# B&R Automation Studio project Nitto (part 14)

#### FB_WebbufferCtrl.st
```iecst
(********************************************************************
 * COPYRIGHT -- Microsoft
 ********************************************************************
 * Programm: MAIN
 * Datei: FB_WebbufferCtrl.st
 * Autor: awalz
 * Erstellt: 26. Juni 2014
 ********************************************************************
 * Implementierung des Programms MAIN
 ********************************************************************)

(* TODO: Bitte Kommentar hier einfügen *)
FUNCTION_BLOCK FB_WebbufferCtrl
	axis.bufferaxis(machineaxis := machineaxis, data := data, CONST := CONST, dancer := dancer, tensionoffset := torqueoffset);
	axis.refSwitchConfig(Enable := TRUE, Axis := axis.ctrl.AxisREF);
//	machineaxis();
	dancer();
	axis.ctrl();
	emcy_inputs();
	keys(clk := clk);
	torqueoffset(enable := TRUE, limitvisuneg := -50, limitvisupos := 50);

//	IF (keys.up.LDT.rtrig.Q OR keys.down.LDT.rtrig.Q ) AND axis.bufferaxis.MC_BR_VelocityControl_0.Active THEN
//		axis.bufferaxis.cmd := CONST.AXIS.STOP;(*deaktivierung des FBs Torque*)
//	ELSIF machineaxis.MC_ReadStatus_0.ContinuousMotion THEN
//		axis.bufferaxis.cmd := CONST.AXIS.START;
//	END_IF
	(*aufruf der Action *)

	status.ready := (axis.ctrl.MC_ReadStatus_0.ContinuousMotion OR axis.ctrl.MC_ReadStatus_0.SynchronizedMotion
				OR axis.ctrl.MC_ReadStatus_0.StandStill) AND NOT axis.ctrl.MC_ReadStatus_0.Disabled;
	status(axisState := axis.ctrl.MC_ReadStatus_0);
	IF axis.ctrl.BasicControl.AxisState.Homed AND (axis.ctrl.MC_ReadStatus_0.StandStill OR axis.ctrl.MC_ReadStatus_0.ContinuousMotion) THEN
		keys.home.LDT.aktion := CONST.LAMP.ON;
	ELSIF axis.ctrl.MC_ReadStatus_0.Disabled THEN
		keys.home.LDT.aktion := CONST.LAMP.BLINK1000;
	ELSIF axis.ctrl.MC_ReadStatus_0.Errorstop THEN
		keys.home.LDT.aktion := CONST.LAMP.BLINK200;
	END_IF
	IF axis.ctrl.MC_ReadStatus_0.Errorstop  AND keys.up.LDT.button AND keys.down.LDT.button THEN
		axis.ctrl(cmd := CONST.AXIS.RESET);
	END_IF
	IF (NOT emcy_inputs.EMCY_Door1 OR NOT emcy_inputs.EMCY_Door2 OR NOT emcy_inputs.EMCY_Door3 OR NOT safety.RequestSTO
		OR NOT emcy_inputs.EMCY_Door4 OR NOT emcy_inputs.EMCY_Door5 OR NOT emcy_inputs.EMCY_Door6) AND NOT  axis.ctrl.MC_ReadStatus_0.Disabled THEN
		axis.ctrl(cmd := CONST.AXIS.POWER_OFF);
		axis.bufferaxis.cmd := CONST.AXIS.STOP;
		mechbrakeON_OFF := FALSE;
	ELSIF  emcy_inputs.EMCY_Door1 AND emcy_inputs.EMCY_Door2 AND emcy_inputs.EMCY_Door3 AND emcy_inputs.EMCY_Door4 AND
		emcy_inputs.EMCY_Door5 AND emcy_inputs.EMCY_Door6 AND axis.ctrl.MC_ReadStatus_0.Disabled AND safety.RequestSTO THEN
		axis.ctrl(cmd := CONST.AXIS.POWER_ON);
		mechbrakeON_OFF := TRUE;

	END_IF
	(* Signal um zu Joggen siehe Mastermodul ac_manual*)
	IF emcy_inputs.EMCY_Door1 AND emcy_inputs.EMCY_Door2 AND emcy_inputs.EMCY_Door3 AND emcy_inputs.EMCY_Door4 AND
		emcy_inputs.EMCY_Door5 AND emcy_inputs.EMCY_Door6 THEN
		emcy_inputs.EMCY_DoorsClosed := TRUE;
	ELSE
		emcy_inputs.EMCY_DoorsClosed := FALSE;
	END_IF

CASE StateCtrl OF
	CTRL_FIRST_START:
		busy := TRUE;
		(*axis.bufferaxis.*)
		StateCtrl := CTRL_EMERGENCYSTOP_BEFORE;

	CTRL_MANUAL_BEFORE://10

		IF BetrCtrl.value = CONST.MACHINEMODES.MANUAL THEN
			BetrStatus(set := TRUE,value := CONST.MACHINEMODES.MANUAL);
			busy := FALSE;
			err(reset := TRUE);
			timer(IN:= FALSE);
			state := ST_IDLE;
			firstStart := TRUE;
			brakeholddelay(PT := T#2s);
			IF axis.ctrl.MC_ReadStatus_0.StandStill THEN
				brakeholddelay.IN:= TRUE;
			END_IF

			IF brakeholddelay.Q AND NOT mechbrakeON_OFF THEN
				brakeholddelay(IN:= FALSE);
				mechbrakeON_OFF := TRUE;
				StateCtrl := CTRL_MANUAL;
			ELSIF mechbrakeON_OFF THEN//25.03.15
				StateCtrl := CTRL_MANUAL;
			END_IF
		ELSIF BetrCtrl.value = CONST.MACHINEMODES.EMERGENCYSTOP THEN
			StateCtrl := CTRL_EMERGENCYSTOP_BEFORE;
		ELSIF BetrCtrl.value = CONST.MACHINEMODES.SAFETYSTOP THEN
			StateCtrl := CTRL_SAFETYSTOP_BEFORE;
		ELSIF BetrCtrl.value = CONST.MACHINEMODES.AUTOMATIC THEN
			StateCtrl := CTRL_AUTO_BEFORE;
		END_IF

	CTRL_MANUAL:
		IF BetrCtrl.value <> CONST.MACHINEMODES.MANUAL THEN
			err(reset := TRUE);
			busy := TRUE;
			StateCtrl := CTRL_MANUAL_AFTER;
		ELSE
			ac_manualbufferCtrl;
			IF axis.ctrl.BasicControl.AxisState.Homed THEN
				 acBuffercyclic; (* Aufruf der Aktion nur wenn die Achse referenziert ist 04.12.14*)
			END_IF
		END_IF

	CTRL_MANUAL_AFTER:

		 acSetModeAfterBuffer;

	CTRL_AUTO_BEFORE:
		IF BetrCtrl.value = CONST.MACHINEMODES.AUTOMATIC THEN
			BetrStatus(set := TRUE, value := CONST.MACHINEMODES.AUTOMATIC);
			(*clamp.init(clk := clk);
			chkStatus.enable := TRUE;*)
			err(reset := TRUE);
			busy := FALSE;
			state := ST_IDLE;
			brakeholddelay(PT := T#2s);
			IF axis.ctrl.MC_ReadStatus_0.StandStill THEN
				brakeholddelay.IN:= TRUE;
			END_IF
			IF brakeholddelay.Q AND NOT mechbrakeON_OFF THEN
				brakeholddelay(IN:= FALSE);
				mechbrakeON_OFF := TRUE;
				StateCtrl := CTRL_AUTO;
			ELSIF mechbrakeON_OFF THEN//25.03.15
				StateCtrl := CTRL_AUTO;
			END_IF
		ELSIF BetrCtrl.value = CONST.MACHINEMODES.EMERGENCYSTOP THEN
			StateCtrl := CTRL_EMERGENCYSTOP_BEFORE;
		ELSIF BetrCtrl.value = CONST.MACHINEMODES.SAFETYSTOP THEN
			StateCtrl := CTRL_SAFETYSTOP_BEFORE;
		ELSIF BetrCtrl.value = CONST.MACHINEMODES.MANUAL THEN
			StateCtrl := CTRL_MANUAL_BEFORE;
		END_IF

	(* ******************************** *)
	(* *********** AUTO *************** *)
	(* ******************************** *)
	CTRL_AUTO:
		IF BetrCtrl.value <> CONST.MACHINEMODES.AUTOMATIC THEN
			err(reset := TRUE);
			busy := TRUE;
			StateCtrl := CTRL_AUTO_AFTER;
		ELSE
			IF axis.ctrl.BasicControl.AxisState.Homed THEN
				 acBuffercyclic; (* Aufruf der Aktion nur wenn die Achse referenziert ist 04.12.14*)
			END_IF
			(*ac_automatic();*)
		END_IF

	CTRL_AUTO_AFTER:
		(*chkStatus.enable := FALSE;*)
		acSetModeAfterBuffer;

	CTRL_STOP_BEFORE:
		IF BetrCtrl.value = CONST.MACHINEMODES.EMERGENCYSTOP THEN
			StateCtrl := CTRL_EMERGENCYSTOP_BEFORE;
		ELSIF BetrCtrl.value = CONST.MACHINEMODES.SAFETYSTOP THEN
			StateCtrl := CTRL_SAFETYSTOP_BEFORE;
		ELSE
			state := ST_IDLE;
			StateCtrl := CTRL_STOP;
		END_IF

	CTRL_STOP:
		IF BetrCtrl.value = CONST.MACHINEMODES.EMERGENCYSTOP THEN
			StateCtrl := CTRL_EMERGENCYSTOP_BEFORE;
		ELSIF BetrCtrl.value = CONST.MACHINEMODES.SAFETYSTOP THEN
			StateCtrl := CTRL_SAFETYSTOP_BEFORE;
		ELSE
			CASE state OF
			ST_IDLE:
				state := ST_QUIT;

			ST_QUIT:
				state := ST_IDLE;
				StateCtrl := CTRL_STOP_AFTER;
			END_CASE
		END_IF

	CTRL_STOP_AFTER:
		IF BetrCtrl.value = CONST.MACHINEMODES.EMERGENCYSTOP THEN
			StateCtrl := CTRL_EMERGENCYSTOP_BEFORE;
		ELSIF BetrCtrl.value = CONST.MACHINEMODES.SAFETYSTOP THEN
			StateCtrl := CTRL_SAFETYSTOP_BEFORE;
		ELSIF BetrCtrl.value = CONST.MACHINEMODES.MANUAL THEN
			StateCtrl := CTRL_MANUAL_BEFORE;
		ELSIF BetrCtrl.value = CONST.MACHINEMODES.AUTOMATIC THEN
			StateCtrl := CTRL_AUTO_BEFORE;
		END_IF

	CTRL_RESET_START:
		BetrStatus.set := TRUE;
		BetrStatus.value := CONST.MACHINEMODES.RESET;
		IF BetrCtrl.value = CONST.MACHINEMODES.EMERGENCYSTOP THEN
			StateCtrl := CTRL_EMERGENCYSTOP_BEFORE;
		ELSIF BetrCtrl.value = CONST.MACHINEMODES.SAFETYSTOP THEN
			StateCtrl := CTRL_SAFETYSTOP_BEFORE;
		ELSE
			IF axis.ctrl.busy  OR axis.ctrl.cmd <> CONST.AXIS.NOACTION THEN
			(*	axis.ctrl(cmd := CONST.AXIS.NOACTION);*)
			ELSE
				mechbrakeON_OFF := FALSE;
				axis.ctrl(cmd := CONST.AXIS.RESET);
				StateCtrl := CTRL_RESET;
			END_IF
		END_IF

	CTRL_RESET:
		axis.ctrl();
		IF BetrCtrl.value = CONST.MACHINEMODES.EMERGENCYSTOP THEN
			StateCtrl := CTRL_EMERGENCYSTOP_BEFORE;
		ELSIF BetrCtrl.value = CONST.MACHINEMODES.SAFETYSTOP THEN
			StateCtrl := CTRL_SAFETYSTOP_BEFORE;
		ELSE
			(*IF NOT unwinderaxis.busy THEN*)
				mechbrakeON_OFF := FALSE;

				axis.ctrl(cmd := CONST.AXIS.POWER_OFF);
				StateCtrl := CTRL_RESET_AFTER;
			(*END_IF*)
		END_IF

	CTRL_RESET_AFTER:
		IF BetrCtrl.value = CONST.MACHINEMODES.RESET THEN
			busy := FALSE;
		ELSE
			busy := TRUE;
			(*clamp.init(clk := clk);
			err.reset();*)
			err(reset := TRUE);
			IF BetrCtrl.value = CONST.MACHINEMODES.EMERGENCYSTOP THEN
				StateCtrl := CTRL_EMERGENCYSTOP_BEFORE;
			ELSIF BetrCtrl.value = CONST.MACHINEMODES.SAFETYSTOP THEN
				StateCtrl := CTRL_SAFETYSTOP_BEFORE;
			ELSIF BetrCtrl.value = CONST.MACHINEMODES.MANUAL THEN
				supplydelay(IN:= TRUE, PT := T#8s);
				IF supplydelay.Q THEN
					axis.ctrl(cmd := CONST.AXIS.POWER_ON);
					busy := TRUE;
					supplydelay(IN:= FALSE);
					StateCtrl := CTRL_MANUAL_BEFORE;
				END_IF
			ELSIF BetrCtrl.value = CONST.MACHINEMODES.AUTOMATIC THEN
				supplydelay(IN:= TRUE, PT := T#8s);
				IF supplydelay.Q THEN
					axis.ctrl(cmd := CONST.AXIS.POWER_ON);
					busy := TRUE;
					supplydelay(IN:= FALSE);
					StateCtrl := CTRL_AUTO_BEFORE;
				END_IF
			END_IF
		END_IF

	CTRL_SAFETYSTOP_BEFORE:
		IF BetrCtrl.value = CONST.MACHINEMODES.EMERGENCYSTOP THEN
			StateCtrl := CTRL_EMERGENCYSTOP_BEFORE;
		ELSE
//			BetrStatus.set := TRUE;
//			BetrStatus.value := CONST.MACHINEMODES.SAFETYSTOP;
//			mechbrakeON_OFF := FALSE;
//			axis.ctrl(cmd := CONST.AXIS.POWER_OFF);(* neue weil die Achse nicht ausgeschaltet wird*)
//			mechbrakeON_OFF := FALSE;
//			state := ST_IDLE;
//			StateCtrl := CTRL_SAFETYSTOP;
			mechbrakeON_OFF := FALSE;
			BetrStatus(set := TRUE,value := CONST.MACHINEMODES.SAFETYSTOP);
			state := ST_IDLE;
			axis.bufferaxis.cmd := CONST.AXIS.STOP;
			axis.ctrl.verzoegerung := 42000.0;
			axis.ctrl.cmd := CONST.AXIS.STOP;
			StateCtrl := CTRL_SAFETYSTOP;
		END_IF

	CTRL_SAFETYSTOP:
		IF BetrCtrl.value = CONST.MACHINEMODES.EMERGENCYSTOP THEN
			StateCtrl := CTRL_EMERGENCYSTOP_BEFORE;
		ELSE
//			CASE state OF
//			ST_IDLE:
//				mechbrakeON_OFF := FALSE;
//			(*	axis.ctrl.cmd := CONST.AXIS.RESET;*)
//				state := ST_QUIT;
//			ST_QUIT:
//				state := ST_QUIT;
//			(*	axis.ctrl(cmd := CONST.AXIS.RESET);*)
//				StateCtrl := CTRL_SAFETYSTOP_AFTER;
//			END_CASE
			IF axis.bufferaxis.MC_ReadStatus_0.StandStill OR axis.bufferaxis.MC_ReadStatus_0.Disabled  THEN
				axis.ctrl.cmd := CONST.AXIS.POWER_OFF;
				StateCtrl := CTRL_SAFETYSTOP_AFTER;
			END_IF
		END_IF

	CTRL_SAFETYSTOP_AFTER:
		busy := FALSE;
		IF BetrCtrl.value = CONST.MACHINEMODES.EMERGENCYSTOP THEN
			busy := TRUE;
			StateCtrl := CTRL_EMERGENCYSTOP_BEFORE;
		ELSIF BetrCtrl.value = CONST.MACHINEMODES.MANUAL THEN
			supplydelay(IN:= TRUE, PT := T#8s);
				IF supplydelay.Q THEN
					axis.ctrl(cmd := CONST.AXIS.POWER_ON);
					busy := TRUE;
					supplydelay(IN:= FALSE);
					StateCtrl := CTRL_MANUAL_BEFORE;
				END_IF
		ELSIF BetrCtrl.value = CONST.MACHINEMODES.AUTOMATIC THEN
				supplydelay(IN:= TRUE, PT := T#8s);
				IF supplydelay.Q THEN
					axis.ctrl(cmd := CONST.AXIS.POWER_ON);
					busy := TRUE;
					supplydelay(IN:= FALSE);
					StateCtrl := CTRL_AUTO_BEFORE;
				END_IF
		END_IF

	CTRL_EMERGENCYSTOP_BEFORE:
//		axis.ctrl(cmd := CONST.AXIS.RESET);
//		mechbrakeON_OFF := FALSE;
//		BetrStatus(set := TRUE,value := CONST.MACHINEMODES.EMERGENCYSTOP);
//		busy := FALSE;
//		StateCtrl := CTRL_EMERGENCYSTOP;
		BetrStatus(set := TRUE,value := CONST.MACHINEMODES.EMERGENCYSTOP);
		mechbrakeON_OFF := FALSE;
		axis.ctrl.verzoegerung:= 1666666; (*200m/min in 2 sek*)
		axis.ctrl.cmd := CONST.AXIS.STOP;
		StateCtrl := CTRL_EMERGENCYSTOP;

	CTRL_EMERGENCYSTOP:
		IF BetrCtrl.value = CONST.MACHINEMODES.EMERGENCYSTOP THEN
			IF axis.ctrl.MC_ReadStatus_0.StandStill OR axis.ctrl.MC_ReadStatus_0.Disabled  THEN
				axis.ctrl.cmd := CONST.AXIS.POWER_OFF;
			END_IF
		ELSE
			busy := TRUE;
			timer(IN := TRUE, PT := T#2s);
			StateCtrl := CTRL_EMERGENCYSTOP_AFTER;
		END_IF

	CTRL_EMERGENCYSTOP_AFTER:
		timer();
		IF BetrCtrl.value = CONST.MACHINEMODES.EMERGENCYSTOP THEN
			timer(IN := FALSE);
			BetrStatus(set := TRUE,value := CONST.MACHINEMODES.EMERGENCYSTOP);
			busy := FALSE;
			StateCtrl := CTRL_EMERGENCYSTOP;
		ELSIF timer.Q THEN
			timer(IN := FALSE);
			StateCtrl := CTRL_RESET_START;
		END_IF

	ELSE
		;
	END_CASE
END_FUNCTION_BLOCK
```

#### FB_WEBBUFFER.st
```iecst
(********************************************************************
 * COPYRIGHT -- Microsoft
 ********************************************************************
 * Programm: MAIN
 * Datei: FB_WEBBUFFER.st
 * Autor: awalz
 * Erstellt: 26. Juni 2014
 ********************************************************************
 * Implementierung des Programms MAIN
 ********************************************************************)

(* TODO: Bitte Kommentar hier einfügen *)
FUNCTION_BLOCK FB_WEBBUFFER
END_FUNCTION_BLOCK
```

#### FB_Bufferaxis.st
```iecst
(********************************************************************
 * COPYRIGHT -- Microsoft
 ********************************************************************
 * Programm: MAIN
 * Datei: NeuerFunktionsBlock.st
 * Autor: awalz
 * Erstellt: 10. Juli 2014
 ********************************************************************
 * Implementierung des Programms MAIN
 ********************************************************************)

(* TODO: Bitte Kommentar hier einfügen *)
FUNCTION_BLOCK FB_Bufferaxis
END_FUNCTION_BLOCK
```

#### FB_BufferConfig.st
```iecst
(********************************************************************
 * COPYRIGHT -- Microsoft
 ********************************************************************
 * Programm: MAIN
 * Datei: FB_BufferConfig.st
 * Autor: awalz
 * Erstellt: 10. Juli 2014
 ********************************************************************
 * Implementierung des Programms MAIN
 ********************************************************************)

(* TODO: Bitte Kommentar hier einfügen *)
FUNCTION_BLOCK FB_BufferConfig

		(*axis.refSwitchConfig(Enable := TRUE, Axis := axis.ctrl.AxisREF);*)
		axis.ctrl.BasicControl.Parameter.Deceleration := 1000;
		axis.ctrl.BasicControl.Parameter.Acceleration := 1000;
		pAxis ACCESS axis.ctrl.AxisREF;
		axis.ctrl();

CASE state OF
	ST_IDLE:
		IF cmd <> CONST.CUTTINGUNIT.CMDs.NO_CMD THEN
			busy := TRUE;
			err(reset := TRUE);
			cmdtmp := cmd;
			IF cmd = CONST.CUTTINGUNIT.CMDs.ABORT THEN
				state := ST_ABORT;
			ELSE
				IF cmd = CONST.CUTTINGUNIT.CMDs.CALIBR THEN
					state := ST_INIT_START;
				ELSIF cmd = CONST.CUTTINGUNIT.CMDs.MOVEFW OR cmd = CONST.CUTTINGUNIT.CMDs.MOVEBW THEN
					state := ST_MOVE_START;
//				ELSE
//					busy := FALSE;
//					err.reset();
				END_IF
			END_IF
		END_IF
//

	(*ST_SET_MODULO:*)

	ST_INIT_START:
		axis();
		IF NOT axis.ctrl.MC_ReadStatus_0.Disabled THEN
			axis.ctrl.cmd := CONST.AXIS.POWER_OFF;
		ELSE
			axis.ctrl.cmd := CONST.AXIS.NOACTION;
			IF NOT axis.ctrl.busy AND  axis.ctrl.MC_ReadStatus_0.Disabled THEN
				pAxis.dig_in.level.neg_hw_end := ncACTIV_HI + ncFORCE;
				pAxis.dig_in.level.pos_hw_end := ncACTIV_HI + ncFORCE;
				InitAxisSubjectPar.Axis := axis.ctrl.AxisREF;
				InitAxisSubjectPar.Subject := ncDIG_IN;
				InitAxisSubjectPar.Execute := TRUE;
				InitAxisSubjectPar();
				IF InitAxisSubjectPar.Done THEN
				(*	axis.refSwitchConfig(Enable := TRUE);*)
				(*	axis.refSwitchConfig.Axis := axis.ctrl.AxisREF;*)
					InitAxisSubjectPar.Execute := FALSE;
					state := ST_REF_START;
				ELSIF InitAxisSubjectPar.Error THEN
					err.text := 'Parameter ncDIG_IN nicht initialisiert';
					err.state := state;
					state := ST_ERROR;
				END_IF
			END_IF
		END_IF

	ST_REF_START:
		InitAxisSubjectPar();
		(*axis.refSwitchConfig();*)
		IF axis.ctrl.MC_ReadStatus_0.Disabled THEN
			axis.ctrl.cmd := CONST.AXIS.POWER_ON;
		ELSIF NOT axis.ctrl.busy AND axis.ctrl.MC_ReadStatus_0.StandStill THEN
		(*	axis.refSwitchConfig(Enable := TRUE);*)
			axis.ctrl.BasicControl.Parameter.HomeMode := mcHOME_LIMIT_SWITCH;
			axis.ctrl.cmd := CONST.AXIS.CALIBR; (* Achse referenzieren*)
			state := ST_CALIBR_WAIT;
		END_IF

	ST_CALIBR_WAIT:
	(*	axis.refSwitchConfig();*)
		IF axis.ctrl.BasicControl.AxisState.Homed THEN
			(*axis.refSwitchConfig(Enable := FALSE);*)
			cmd := CONST.CUTTINGUNIT.CMDs.NO_CMD;
			axis.ctrl(cmd := CONST.AXIS.NOACTION);
			status.ready := TRUE;
			cmdtmp := cmd;
			state := ST_QUIT;(* Achse ist referenziert*)
		(*	state := ST_CALIBR_START_NULLPOS;*)
		ELSIF cmd <> CONST.CUTTINGUNIT.CMDs.CALIBR THEN
			axis.ctrl(cmd := CONST.AXIS.STOP);
			state := ST_QUIT;
		END_IF

	ST_MOVE_START:
//		masterAxis.ctrl.ref.ReadStatus();
		IF cmd = CONST.CUTTINGUNIT.CMDs.NO_CMD THEN
			busy := FALSE;
			state := ST_IDLE;
		ELSE
			IF cmd = CONST.CUTTINGUNIT.CMDs.MOVEBW THEN
				axis.ctrl.velocity	:= 0.01;
				axis.ctrl.cmd := CONST.AXIS.JOG_NEG;
				state := ST_MOVE_WAIT;
			ELSE
				axis.ctrl.velocity := 0.02;
				axis.ctrl.cmd := CONST.AXIS.JOG_POS;
				state := ST_MOVE_WAIT;
			END_IF

		END_IF

	ST_MOVE_WAIT:
		axis.ctrl();
		IF cmd = CONST.CUTTINGUNIT.CMDs.NO_CMD THEN
			axis.ctrl(cmd := CONST.AXIS.NOACTION );
			state := ST_MOVE_QUIT;
		END_IF
//
	ST_MOVE_QUIT: (* hier evtl. koppeln*)
		state := ST_QUIT;

	ST_ERROR:
		IF LEN(err.fnc) < 1 THEN
			err.fnc := 'FB_CuttingConfig';
		END_IF
		err(flag := TRUE);
		state := ST_QUIT;

	ST_ABORT:
		state := ST_ABORT_QUIT;

	ST_ABORT_QUIT:
		busy := FALSE;
		IF cmd <> CONST.CUTTINGUNIT.CMDs.NO_CMD THEN
			state := ST_IDLE;
		END_IF

	ST_QUIT:
		IF cmd = CONST.CUTTINGUNIT.CMDs.ABORT THEN
			busy := TRUE;
			state := ST_ABORT;
		ELSE
			busy := FALSE;
			IF cmd = CONST.CUTTINGUNIT.CMDs.NO_CMD THEN
				axis.ctrl(cmd := CONST.AXIS.NOACTION);
				state := ST_IDLE;
			END_IF
		END_IF

	END_CASE
//InitAxisSubjectPar();
END_FUNCTION_BLOCK
```

#### FB_TorqueAxis.st
```iecst
(********************************************************************
 * COPYRIGHT -- Microsoft
 ********************************************************************
 * Programm: MAIN
 * Datei: FB_TorqueAxis.st
 * Autor: awalz
 * Erstellt: 11. Juli 2014
 ********************************************************************
 * Implementierung des Programms MAIN
 ********************************************************************)

(* TODO: Bitte Kommentar hier einfügen *)
FUNCTION_BLOCK FB_TorqueAxis
	(********************MC_BR_READDRIVESTATUS***********************)
	MC_BR_ReadDriveStatus_0.Enable := NOT(MC_BR_ReadDriveStatus_0.Error);
	MC_BR_ReadDriveStatus_0.Axis := AxisREF;
	MC_BR_ReadDriveStatus_0.AdrDriveStatus := ADR(BasicControl.Status.DriveStatus);
	MC_BR_ReadDriveStatus_0();
	(************************ MC_READSTATUS *************************)
	MC_ReadStatus_0.Enable :=  NOT MC_ReadStatus_0.Error;
	MC_ReadStatus_0.Axis := AxisREF;
	MC_ReadStatus_0();
	//*****************************************************************
	IF enablemerker THEN
		MC_TorqueControl_0.Execute := TRUE;(*wieder einschalten*)
		enablemerker := FALSE;
	END_IF
	IF MC_TorqueControl_0.Torque <> settorque OR MC_TorqueControl_0.Velocity <> setvelocity AND MC_TorqueControl_0.Active THEN
		MC_TorqueControl_0.Execute := FALSE;
		enablemerker := TRUE;
	END_IF

	MC_TorqueControl_0.TorqueRamp 	:= 1;
	MC_TorqueControl_0.Velocity 	:= setvelocity; (*300;*)
	MC_TorqueControl_0.Acceleration := 1000;
	MC_TorqueControl_0.Axis			:= AxisREF;
	MC_TorqueControl_0.Torque 		:= settorque;

	IF MC_TorqueControl_0.Execute AND MC_TorqueControl_0.CommandAborted AND cmdtmp = CONST.AXIS.START THEN
		MC_TorqueControl_0.Execute := FALSE;
	ELSIF NOT MC_TorqueControl_0.Execute  AND cmdtmp = CONST.AXIS.POWER_ON AND NOT MC_TorqueControl_0.Error AND MC_ReadStatus_0.StandStill THEN
		MC_TorqueControl_0.Execute := TRUE;
	ELSIF MC_TorqueControl_0.Error AND cmdtmp = CONST.AXIS.START THEN
		MC_TorqueControl_0.Execute := FALSE;
	END_IF
	IF NOT( MC_ReadStatus_0.StandStill OR MC_ReadStatus_0.ContinuousMotion OR MC_ReadStatus_0.DiscreteMotion OR MC_ReadStatus_0.SynchronizedMotion) THEN
			MC_TorqueControl_0.Execute := FALSE;
	END_IF

	IF 	cmd = CONST.AXIS.START AND NOT MC_TorqueControl_0.InTorque THEN
		MC_Stop_0.Execute := FALSE;
		MC_TorqueControl_0.Execute := TRUE;
		cmdtmp := cmd;
		cmd:= CONST.AXIS.NOACTION;
	END_IF
	//********************************************************************
	MC_Stop_0.Deceleration	:= 2000;
	IF cmd = CONST.AXIS.STOP THEN
		IF  MC_ReadStatus_0.ContinuousMotion OR MC_ReadStatus_0.DiscreteMotion THEN
				MC_TorqueControl_0.Execute := FALSE;
				MC_Stop_0.Execute := TRUE;
		END_IF
		IF MC_Stop_0.Done THEN
			MC_Stop_0.Execute := FALSE;
			cmdtmp := cmd;
			cmd := CONST.AXIS.NOACTION;
		END_IF
	END_IF
	(***************************************************************
        FUNCTION Block Calls
	(************************** MC_STOP *****************************)
	MC_Stop_0.Axis := AxisREF;
	MC_Stop_0();
	IF BasicControl.Status.DriveStatus.NetworkInit THEN
		MC_TorqueControl_0();
	END_IF
//	(************************** MC_POWER ****************************)
//	MC_Power_0.Axis := AxisREF;  (* pointer to axis *)
//	MC_Power_0(); (*Laut B& R darf man den FB nicht zwei mal für die selbe Achse aufrufen*)
	(************************** MC_RESET ****************************)
//	MC_Reset_0.Axis := AxisREF;
//	MC_Reset_0();
END_FUNCTION_BLOCK
```

#### FB_BufferTensionCtrl.st
```iecst
(********************************************************************
 * COPYRIGHT -- Microsoft
 ********************************************************************
 * Programm: MAIN
 * Datei: FB_BufferTensionCtrl.st
 * Autor: awalz
 * Erstellt: 21. November 2014
 ********************************************************************
 * Implementierung des Programms MAIN
 ********************************************************************)

(* TODO: Bitte Kommentar hier einfügen *)
FUNCTION_BLOCK FB_BufferTensionCtrl
	IF firststart THEN
		pAxis ACCESS AxisREF;
		LCRPIDpara_0.Kfbk					:= 2.0; // Anti-windup used
		LCRPIDpara_0.d_mode					:= LCRPID_D_MODE_E;	// differentiate control deviation
		LCRPIDpara_0.fbk_mode				:= LCRPID_FBK_MODE_INTERN;	// feedback of internal output
		LCRPID_0.mode						:= LCRPID_MODE_AUTO;	// Standard PID operating mod
		// 50.000 = 3 m/min
		LCRPID_0.Y_max						:= 100;	// percent
		LCRPID_0.Y_min						:= -100;// percent

		LCRPIDpara_0.Kp						:= 3; (*11*)
		LCRPIDpara_0.Tn						:= 1.1;	// Integrative part
		LCRPIDpara_0.Tv						:= 0.0; // D-part
		LCRPIDpara_0.Tf						:= 0;(*0.020;*)
		LCRPIDpara_0.WX_max					:= 1000.0;
		LCRPIDpara_0.WX_min					:= -1000.0;
//		LCRPIDpara_0.deadband				:= 10;
//		LCRPIDpara_0.deadband_mode			:= LCRPID_DEADBAND_MODE_STANDARD;
		LCRPID_0.ident						:= LCRPIDpara_0.ident;
		// Maximum controller output:

		//set filter time for tension sensor
		LCRPT1e_ActTension.V		:= 1.0;
		LCRPT1e_ActTension.T1		:= TENSION_T_FILTER;(*0.2*)
		LCRPT1e_ActTension.enable	:= TRUE;
//		vecD[0]		:= 80;		// [mm]
//		vecD[1]		:= 1200.0;		// [mm]
//		vecD[2]		:= 0.0;
//		vecKV[0]	:= 2.7;	// [As]
//		vecKV[1]	:= 80.0;	// [As]
//		vecKV[2]	:= 0.0;
//		vecTN[0]	:= 0.00;	// [s]
//		vecTN[1]	:= 0.15;	// [s]
//		vecTN[2]	:= 0.0;
//		WNCLipSctrlPara_Unwinder.pSysPara		:= ADR(UnwinderSysPara);
//		WNCLipSctrlPara_Unwinder.numPoints		:= 2;
//		WNCLipSctrlPara_Unwinder.pVecDiam		:= ADR(vecD);
//		WNCLipSctrlPara_Unwinder.pVecSctrlKV	:= ADR(vecKV);
//		WNCLipSctrlPara_Unwinder.pVecSctrlTN	:= ADR(vecTN)
		//**************	set parameters for speed controller **************

		MC_BR_VelocityControl_0.Acceleration	:= 20000; (*1000000 wo kommt der astronomischer Wert her*)
		MC_BR_VelocityControl_0.Deceleration	:= 20000;
		MC_BR_VelocityControl_0.TorqueMode		:= mcLIMIT;
		MC_BR_VelocityControl_0.SctrlKv 		:= 0.1;
		MC_BR_VelocityControl_0.SctrlTn			:= 0.15;

	(*	MC_BR_TorqueControl_0.Acceleration		:= 100000;*)

		//***********************************************************************
		firststart := FALSE;
	 END_IF
	//************************** LCRPIDpara *******************************
	//lowpass filter for sensor signal
	LCRPT1e_ActTension.x		:=  dancer.tension_scaled; (*.IO.AIn.FlengeDMS.Value.Scaled;*)
	LCRPT1e_ActTension();
	LCRPIDpara_0();
	//************************** LCRPID *******************************
	LCRPID_0.ident						:= LCRPIDpara_0.ident;
	// PID controller:

	//  setpoint  		"W" = web tension from application recipe
	//  actual value	"X" = measured web tension from flenge DMS input (*override wird beim füllen draufgegebe*)
	LCRPID_0.W			:= LIMIT (0, data.recipe.SetTension + tensionoffset.setvalueVisu + override, 200);
//	LCRPID_0.X			:= floor (LCRPT1e_ActTension.y);
	LCRPID_0.X			:= LCRPT1e_ActTension.y;
	LCRPID_0();
	(*OutPID				:= LCRPID_TM.Y * TM_SCALE_PID_OUT_TO_OFFSET;*)
	CyclicVelocity		:= LCRPID_0.Y * TM_SCALE_PID_OUT_TO_OFFSET;

	IF CyclicVelocity < -1 THEN
		MC_BR_VelocityControl_0.CyclicTorque :=  -1 * settorque ;
	ELSE
		MC_BR_VelocityControl_0.CyclicTorque :=  settorque;
	END_IF
	// ================
	// CHECK ERRORS
	// ================

	IF (LCRPID_0.status > 12022) AND
	   (LCRPID_0.status < 65534) THEN
//		// Error in PID controller detected -> stop control
		AxisStep		:= ST_CTRL_OFF;
	END_IF

	CASE AxisStep OF
		//********************* INITIALISATION ************************
		ST_INIT1:
			LCRPIDpara_0.enable		:= TRUE;
			LCRPIDpara_0.enter		:= FALSE;
			LCRPID_0.enable			:= FALSE; (* 10.12.14*)
		(*	LCRPID_0.enable			:= FALSE;*)
			MC_BR_VelocityControl_0.Enable := FALSE;
			AxisStep					:= ST_READY;

		//********************* WAIT FOR COMMANDS ************************
		ST_READY:
		(*	MC_BR_CyclicWrite_0.Enable			:= FALSE;*)
			IF cmd = CONST.AXIS.START  THEN
				(*TensMeas.Command.startTmControl	:= FALSE;*)
			(*	MC_BR_CyclicWrite_0.Enable		:= TRUE;*)
				LCRPID_0.enable			:= FALSE;
				AxisStep		:= ST_WAIT_POWER_ENABLED;
			ELSIF cmd = CONST.AXIS.JOG_POS THEN
				AxisStep := ST_MOVE_POS;
			ELSIF cmd = CONST.AXIS.JOG_NEG THEN
				AxisStep := ST_MOVE_NEG;
			END_IF
			// End of STEP_TM_READY
		//********************* WAIT FOR DRIVES BEING ENABLED ************************
		ST_WAIT_POWER_ENABLED:
			IF  MC_ReadStatus_0.StandStill OR  MC_ReadStatus_0.ContinuousMotion THEN
				AxisStep			:= ST_LOAD_PARA_START;
				// Generate rising edge at the enter input in order to update
				// PID controller parameters
				LCRPIDpara_0.enter	:= FALSE;
			ELSIF MC_ReadStatus_0.Error THEN
				AxisStep := ST_INIT1;
			END_IF
			// End of STEP_TM_WAIT_POWER_ENABLED
		//********************* START PARAMETER LOADING ************************
		ST_LOAD_PARA_START:
			// Rising edge for updating controller parameter
			LCRPIDpara_0.enter		:= TRUE;
			AxisStep				:= ST_WAIT_LOAD_PARA_DONE;
//		//********************* WAIT FOR PARAMETER LOAD COMPLETE ************************
		ST_WAIT_LOAD_PARA_DONE:
			LCRPIDpara_0.enter		:= FALSE;
			AxisStep				:= ST_WAIT_SWITCH_CTRL_ON;
			// End of STEP_TM_WAIT_LOAD_PARA_DONE
//
//		//********************* ACTIVATE CONTROL ************************
		ST_WAIT_SWITCH_CTRL_ON:
			IF  MC_ReadStatus_0.StandStill AND (LCRPIDpara_0.ident <> 0)  THEN
				// Enable PID controller and Offset correction for web tension control
				LCRPID_0.enable				:= TRUE;
//				MC_BR_TorqueControl_0.Enable := TRUE;
//				MC_BR_TorqueControl_0.StartSignal :=TRUE;
				MC_BR_VelocityControl_0.Enable 	:= TRUE;
				AxisStep						:= ST_CTRL_ACTIVE;
			ELSIF MC_ReadStatus_0.ContinuousMotion THEN (* PI_REgler und Achse sind bereits aktiv*)
				MC_BR_VelocityControl_0.Enable 	:= TRUE;
				LCRPID_0.enable					:= TRUE;
				AxisStep						:= ST_CTRL_ACTIVE;

			END_IF
			// Go to ready state in order to update controller parameter
			IF  cmd = CONST.AXIS.STOP  THEN
				AxisStep	:= ST_INIT1;
			END_IF
//			// End of STEP_TM_WAIT_SWITCH_CTRL_ON
//
//		//********************* CONTROL IS ACTIVE ************************
		ST_CTRL_ACTIVE:
			MC_BR_VelocityControl_0.CyclicVelocityCorrection := LIMIT (-300, CyclicVelocity, 300);
		(*		MC_BR_TorqueControl_0.Torque :=  LIMIT (-50, CyclicVelocity, 50);*)
			IF cmd = CONST.AXIS.STOP	OR  MC_ReadStatus_0.Disabled  THEN
			(*	TensMeas.Command.stopTmControl 			:= FALSE;*)
				MC_BR_VelocityControl_0.Enable 	:= FALSE;
//				MC_BR_TorqueControl_0.Enable := FALSE;
//				MC_BR_TorqueControl_0.StartSignal :=FALSE;
			(*	AxisStep	:= ST_CTRL_OFF;*)
				AxisStep := ST_INIT1;
			ELSIF MC_BR_VelocityControl_0.CommandAborted AND cmd = CONST.AXIS.START THEN
				MC_BR_VelocityControl_0.Enable 	:= FALSE;
				AxisStep := ST_INIT1;
			ELSIF  cmd = CONST.AXIS.JOG_POS OR cmd = CONST.AXIS.JOG_NEG THEN
				MC_BR_VelocityControl_0.Enable 	:= FALSE;
				AxisStep := ST_INIT1;
			END_IF
//		// End of STEP_TM_CTRL_ACTIVE
		ST_MOVE_POS: (* Achse hoch fahren*)
			MC_BR_VelocityControl_0.CyclicVelocityCorrection := LIMIT (-300, CyclicVelocity, 300);
			IF cmd = CONST.AXIS.JOG_POS AND MC_ReadStatus_0.StandStill THEN
				MC_BR_VelocityControl_0.CyclicVelocity := 100;
				MC_BR_VelocityControl_0.Enable := TRUE;
			ELSIF cmd <> CONST.AXIS.JOG_POS THEN
				MC_BR_VelocityControl_0.CyclicVelocity := 0;
				MC_BR_VelocityControl_0.Enable := FALSE;
				AxisStep := ST_INIT1;
			END_IF

		ST_MOVE_NEG: (* Achse runter fahren*)
			MC_BR_VelocityControl_0.CyclicVelocityCorrection := LIMIT (-300, CyclicVelocity, 300);
			IF cmd = CONST.AXIS.JOG_NEG AND MC_ReadStatus_0.StandStill THEN
				MC_BR_VelocityControl_0.CyclicVelocity := - 100;
				MC_BR_VelocityControl_0.Enable := TRUE;
			ELSIF cmd <> CONST.AXIS.JOG_NEG THEN
				MC_BR_VelocityControl_0.CyclicVelocity := 0;
				MC_BR_VelocityControl_0.Enable := FALSE;
				AxisStep := ST_INIT1;
			END_IF
//		//********************* PAUSING CONTROL ************************
		ST_CTRL_PAUSE:
//			action_TmCtrlOff;
//			// Go to step for waiting to enable control again
			IF cmd = CONST.AXIS.START THEN
				AxisStep	:= ST_WAIT_SWITCH_CTRL_ON;
			ELSIF cmd = CONST.AXIS.POWER_OFF THEN
				AxisStep	:= ST_CTRL_OFF;
			END_IF
//			// End of STEP_TM_CTRL_PAUSE
//
//		//********************* SWITCH CONTROL OFF ************************
		ST_CTRL_OFF:
//			action_TmCtrlOff;
//			// Go to step for waiting fo new commands
			AxisStep					:= ST_INIT1;
//			// End of STEP_TM_CTRL_OFF

	END_CASE
	//********************************************************************
	// Function Block Calls
	//*********************************************************************
	//***********************************************************************
	MC_ReadActualPosition_0.Enable := NOT(MC_ReadActualPosition_0.Error);
	MC_ReadActualPosition_0.Axis := AxisREF;
	MC_ReadActualPosition_0();

	MC_BR_ReadDriveStatus_0.Axis			:= AxisREF;
	MC_BR_ReadDriveStatus_0.AdrDriveStatus	:= ADR(BasicControl.Status.DriveStatus); (*DriveStatus;*)
	MC_BR_ReadDriveStatus_0.Enable			:= NOT MC_BR_ReadDriveStatus_0.Error; (*MC_BR_ReadDriveStatus_0.Error;*)
	MC_BR_ReadDriveStatus_0();

//	MC_BR_CyclicWrite_0.Axis		:= AxisREF;
//	MC_BR_CyclicWrite_0.DataAddress	:= ADR(CyclicVelocity);
//	MC_BR_CyclicWrite_0.DataType	:= ncPAR_TYP_REAL;  nicht vergessen in Acps10map ACOPOS Parameter gpbsSPTa mit zschreiben
//	MC_BR_CyclicWrite_0.ParID		:= ACP10PAR_VAR_R4_0 + 0;
//	MC_BR_CyclicWrite_0();
//	MC_BR_TorqueControl_0.Axis := AxisREF;//
// 	MC_BR_TorqueControl_0();//
//	***********************MC_BR_VelocityControl******************
	MC_BR_VelocityControl_0.Axis			:= AxisREF;//
	MC_BR_VelocityControl_0();
	(************************ MC_READSTATUS *************************)
	MC_ReadStatus_0.Enable :=  NOT MC_ReadStatus_0.Error;
	MC_ReadStatus_0.Axis := AxisREF;
	MC_ReadStatus_0();
	(************************** MC_POWER ****************************)
//	MC_Power_0.Axis := AxisREF;  (* pointer to axis *)
//	MC_Power_0();

	(************************** MC_STOP *****************************)
//	MC_Stop_0.Axis := AxisREF;
//	MC_Stop_0();
	(***************************MC_HALT******************************)
	(*MC_Halt_0.Axis := AxisREF;
	MC_Halt_0();
	(************************** MC_RESET ****************************)
//	MC_Reset_0.Axis := AxisREF;
//	MC_Reset_0();
END_FUNCTION_BLOCK
```

#### FB_BUFFER_RECIPE_DATA.st
```iecst
(********************************************************************
 * COPYRIGHT -- Microsoft
 ********************************************************************
 * Programm: MAIN
 * Datei: FB_BUFFER_RECIPE_DATA.st
 * Autor: awalz
 * Erstellt: 26. November 2014
 ********************************************************************
 * Implementierung des Programms MAIN
 ********************************************************************)

(* TODO: Bitte Kommentar hier einfügen *)
FUNCTION_BLOCK FB_BUFFER_RECIPE_DATA
END_FUNCTION_BLOCK
```

#### FB_BUFFER_DATA.st
```iecst
(********************************************************************
 * COPYRIGHT -- Microsoft
 ********************************************************************
 * Programm: MAIN
 * Datei: FB_DataBufferTension.st
 * Autor: awalz
 * Erstellt: 20. November 2014
 ********************************************************************
 * Implementierung des Programms MAIN
 ********************************************************************)

(* TODO: Bitte Kommentar hier einfügen *)
FUNCTION_BLOCK FB_BUFFER_DATA
END_FUNCTION_BLOCK
```

#### Package Logical/MainMachineCtrl/MAIN/Pullbreak - Neues leeres Paket

#### FB_PullBreakUnitConfig.st
```iecst
(********************************************************************
 * COPYRIGHT -- Microsoft
 ********************************************************************
 * Programm: MAIN
 * Datei: FB_PullBreakUnitConfig.st
 * Autor: Awalz
 * Erstellt: 7. Mai 2014
 ********************************************************************
 * Implementierung des Programms MAIN
 ********************************************************************)

 (*<$Description$> TODO: Bitte Kommentar hier einzufügen </$Description$>*)
FUNCTION_BLOCK FB_PullBreakUnitConfig
 axis.cplOn();
 axis.cplOff();
	axis.ctrl.BasicControl.Parameter.Deceleration	:= 80000.0; //only for initialization
	axis.ctrl.BasicControl.Parameter.Acceleration	:= 80000.0;

	CASE state OF
	ST_IDLE:
		IF cmd <> CONST.CUTTINGUNIT.CMDs.NO_CMD THEN
			busy := TRUE;
			err(reset:= TRUE);
			cmdtmp := cmd;
			IF cmd = CONST.CUTTINGUNIT.CMDs.CPL_ON THEN
				cmdtmp := cmd;
				state := ST_CPL_START;
			ELSIF cmd = CONST.CUTTINGUNIT.CMDs.CPL_OFF THEN
				cmdtmp := cmd;
				state := ST_CPLOFF_START;
			ELSIF  cmd =  CONST.CUTTINGUNIT.CMDs.MOVEBW OR cmd = CONST.CUTTINGUNIT.CMDs.MOVEFW THEN
				state := ST_MOVE_START;
			ELSE
				err.state := state;
				err(text := 'CommandError');
				state := ST_ERROR;
			END_IF
		END_IF

	ST_CPL_START:
		axis.ctrl();

		IF cmd = CONST.CUTTINGUNIT.CMDs.ABORT THEN
			state := ST_ABORT;
		ELSIF axis.cplOn.InGear THEN
			status.isCoupled := TRUE;
			status.mode := CONST.UNITMODEs.ENABLE;
			state := ST_QUIT;
		ELSIF axis.cplOn.Busy  THEN
			status.isCoupled := TRUE;
			status.mode := CONST.UNITMODEs.ENABLE;
			state := ST_QUIT;
		ELSIF axis.ctrl.MC_ReadStatus_0.StandStill THEN
			axis.cplOn(Execute := TRUE, Master := machineMasterCtrl.AxisREF, Slave := axis.ctrl.AxisREF,
						Acceleration := 40000, Deceleration := 40000 , RatioDenominator := axis.setGearRatio.ratioDenominator,
						RatioNumerator := axis.setGearRatio.ratioNumeratorOut);
			state := ST_CPL_WAIT;
		END_IF

	ST_CPL_WAIT:
		axis.cplOn( Master := machineMasterCtrl.AxisREF, Slave := axis.ctrl.AxisREF );
		IF axis.cplOn.Busy THEN
			axis.cplOn(Execute := FALSE, Master := machineMasterCtrl.AxisREF, Slave := axis.ctrl.AxisREF);
				status.isCoupled := TRUE;
				status.mode := CONST.UNITMODEs.ENABLE;
				state := ST_QUIT;
		ELSIF axis.cplOn.Error THEN
				err.id := axis.cplOn.ErrorID;
				err.fnc := 'axis.cplOn';
				err.state := state;
				state := ST_ERROR;
(*			ELSIF axis.cplOn.CommandAborted THEN
				err.fnc := 'axis.cplOn CommandAborted';
				err.state := state;
				state := ST_ERROR;
			ELSIF axis.cplOn.InGear THEN *)
		END_IF

	ST_CPLOFF_START:
		IF cmd = CONST.CUTTINGUNIT.CMDs.ABORT THEN
			state := ST_ABORT;
		ELSIF axis.cplOff.Error  THEN
			err.state := state;
			err.text := 'MC_GearOut';
			state := ST_ERROR;
		ELSIF axis.cplOff.Busy OR axis.cplOff.Execute THEN
			axis.cplOff(Execute := FALSE, Slave := axis.ctrl.AxisREF);
		ELSE
			axis.cplOff(Execute := TRUE, Slave := axis.ctrl.AxisREF);
			state := ST_CPLOFF_WAIT;
		END_IF

	ST_CPLOFF_WAIT:
		axis.cplOff( Slave := axis.ctrl.AxisREF );
		IF  axis.cplOff.Done THEN
			IF axis.cplOff.Error THEN
				err.id := axis.cplOff.ErrorID;
				err.fnc := 'axis.cplOff';
				err.state := state;
				state := ST_ERROR;
(*neu 20.08.14*)
			ELSE
				axis.cplOff.Execute := FALSE;
				status.isCoupled := FALSE;
				IF cmd = CONST.CUTTINGUNIT.CMDs.MOVEBW OR cmd = CONST.CUTTINGUNIT.CMDs.MOVEFW THEN
					state := ST_MOVE_START;
				ELSE
				(*	status.mode := CONST.UNITMODEs.DISABLE;*)
					state := ST_QUIT;
				END_IF

			END_IF

		END_IF
//////////20.08.14 Kundenwunsch: um die Zugstation zu reinigen sollte man die joggen können
		ST_MOVE_START:
//		masterAxis.ctrl.ref.ReadStatus();
		IF cmd = CONST.CUTTINGUNIT.CMDs.NO_CMD THEN
			busy := FALSE;
			state := ST_IDLE;
		ELSIF axis.ctrl.MC_ReadStatus_0.SynchronizedMotion THEN
//			err.text := 'MOVE nicht möglich. Achse ist gekoppelt';
//			err.state := state;
			state := ST_CPLOFF_START;
//		ELSIF status.isCalibrated THEN (* die Stanze soll man auch ohne zu rferenzieren drehen können*)
//			IF axis.ctrl.busy (*OR axis.ctrl.cmd <> CONST.AXIS.NOACTION*) THEN
//				axis.ctrl(cmd := CONST.AXIS.NOACTION);
		ELSIF axis.ctrl.MC_ReadStatus_0.StandStill OR axis.ctrl.MC_ReadStatus_0.ContinuousMotion THEN
			IF cmd = CONST.CUTTINGUNIT.CMDs.MOVEBW THEN
				axis.ctrl(cmd := CONST.AXIS.JOG_NEG, velocity := 4);
				state := ST_MOVE_WAIT;
			ELSE
				axis.ctrl(cmd := CONST.AXIS.JOG_POS, velocity := 4);
				state := ST_MOVE_WAIT;
			END_IF
		END_IF

	ST_MOVE_WAIT:
		axis.ctrl();
		IF cmd = CONST.CUTTINGUNIT.CMDs.NO_CMD THEN
			axis.ctrl(cmd := CONST.AXIS.NOACTION );
			state := ST_MOVE_QUIT;
		END_IF
//
	ST_MOVE_QUIT: (* hier evtl. koppeln*)
		state := ST_CPL_START;
		(*state := ST_QUIT;*)

	ST_ERROR:
		IF LEN(err.fnc) < 1 THEN
			err.fnc := 'FB_PullBrakeUnitConfig';
		END_IF
		err.flag := TRUE;
		state := ST_QUIT;

	ST_ABORT:
		state := ST_ABORT_QUIT;

	ST_ABORT_QUIT:
		busy := FALSE;
		IF cmd <> CONST.CUTTINGUNIT.CMDs.NO_CMD THEN
			state := ST_IDLE;
		END_IF

	ST_QUIT:
		IF cmd = CONST.CUTTINGUNIT.CMDs.ABORT THEN
			busy := TRUE;
			state := ST_ABORT;
		ELSE
			busy := FALSE;
			IF cmd = CONST.CUTTINGUNIT.CMDs.NO_CMD THEN
				state := ST_IDLE;
			END_IF
		END_IF
	END_CASE
END_FUNCTION_BLOCK
```

#### ac_setStateAfterPB.st
```iecst
(********************************************************************
 * COPYRIGHT -- Microsoft
 ********************************************************************
 * Programm: MAIN
 * Datei: ac_setStateAfterPB.st
 * Autor: Awalz
 * Erstellt: 7. Mai 2014
 ********************************************************************
 * Implementierung des Programms MAIN
 ********************************************************************)

 (*<$Description$> Fügt eine neue Aktion zum IEC Programm oder Bibliothek </$Description$>*)
ACTION ac_setStateAfterPB:
		IF BetrCtrl.value = CONST.MACHINEMODES.EMERGENCYSTOP THEN
		StateCtrl := CTRL_EMERGENCYSTOP_BEFORE;
	ELSIF BetrCtrl.value = CONST.MACHINEMODES.SAFETYSTOP THEN
		StateCtrl := CTRL_SAFETYSTOP_BEFORE;
	ELSIF BetrCtrl.value = CONST.MACHINEMODES.MANUAL THEN
		StateCtrl := CTRL_STOP_BEFORE;
	ELSIF BetrCtrl.value = CONST.MACHINEMODES.AUTOMATIC THEN
		StateCtrl := CTRL_STOP_BEFORE;
	END_IF
END_ACTION
```

#### FB_PullbreakUnitCtrl.st
```iecst
(********************************************************************
 * COPYRIGHT -- Microsoft
 ********************************************************************
 * Programm: MAIN
 * Datei: FB_PullbrakeUnitCtrl.st
 * Autor: Awalz
 * Erstellt: 27. März 2014
 ********************************************************************
 * Implementierung des Programms MAIN
 ********************************************************************)

(*<$Description$> TODO: Bitte Kommentar hier einzufügen </$Description$>*)
FUNCTION_BLOCK FB_PullbreakUnitCtrl
	axis.ctrl();
	mode := CONST.UNITMODEs.ENABLE;
	chkStatus(setMode := mode, status := status);
	clamp(clk := clk);
	hubctrl(clk := clk);
	status(axisState := axis.ctrl.MC_ReadStatus_0);
	status.ready  := axis.ctrl.MC_ReadStatus_0.SynchronizedMotion;
	emcy_inputs();
	IF emcy_inputs.EMCY_Door1 THEN
		emcy_inputs.EMCY_DoorsClosed := TRUE;
	ELSE
		emcy_inputs.EMCY_DoorsClosed := FALSE;
	END_IF
	axis.setGearRatio(limitvisuneg := -20, limitvisupos := 100, limitrationeg := 800, limitratiopos := 1500);
	IF axis.setGearRatio.enable THEN
	axis.cplOn(RatioNumerator := axis.setGearRatio.ratioNumeratorOut,
			Execute := axis.setGearRatio.trigger ,RatioDenominator := axis.setGearRatio.ratioDenominator,
			Acceleration := 40000, Deceleration := 40000);
	END_IF
	IF axis.ctrl.MC_ReadStatus_0.Errorstop AND panel.LDTRESET.LDT.button THEN
		axis.ctrl.cmd := CONST.AXIS.RESET;
	ELSIF axis.ctrl.MC_ReadStatus_0.Disabled AND panel.LDTRESET.LDT.ftrig.Q AND cmdCtrl.value = CONST.AXIS.NOACTION THEN
		axis.ctrl.cmd := CONST.AXIS.NOACTION;
	END_IF
	safety();

	CASE StateCtrl OF
	CTRL_FIRST_START:
		busy := TRUE;
		(*axis.ctrl.BasicControl.Command.Power := TRUE;*)
		StateCtrl := CTRL_EMERGENCYSTOP_BEFORE;

	CTRL_MANUAL_BEFORE:
		IF BetrCtrl.value = CONST.MACHINEMODES.MANUAL THEN
			clamp.toDown_o := TRUE;(* damit die ZUGstation beim Start unten bleibt*)
			BetrStatus(set := TRUE, value := CONST.MACHINEMODES.MANUAL);
			chkStatus.enable := TRUE;
			err(reset := TRUE);
			busy := FALSE;
			timer(IN:= FALSE);
			state := ST_IDLE;
			manualFirst := TRUE;
			StateCtrl := CTRL_MANUAL;
		ELSIF BetrCtrl.value = CONST.MACHINEMODES.EMERGENCYSTOP THEN
			StateCtrl := CTRL_EMERGENCYSTOP_BEFORE;
		ELSIF BetrCtrl.value = CONST.MACHINEMODES.SAFETYSTOP THEN
			StateCtrl := CTRL_SAFETYSTOP_BEFORE;
		ELSIF BetrCtrl.value = CONST.MACHINEMODES.AUTOMATIC THEN
			StateCtrl := CTRL_AUTO_BEFORE;
		END_IF

	CTRL_MANUAL:
		IF BetrCtrl.value <> CONST.MACHINEMODES.MANUAL THEN
			err(reset := TRUE);
			busy := TRUE;
			StateCtrl := CTRL_MANUAL_AFTER;
	(*ELSIF axis.ctrl.MC_ReadStatus_0.StandStill THEN
				timer(IN := TRUE, PT := T#8s);
				IF timer.Q THEN
					ac_manualPB;
				END_IF*)
		ELSE
			ac_manualPB;
			(*StateCtrl := CTRL_RESET_START;*)
		END_IF

	CTRL_MANUAL_AFTER:
		timer(IN:= FALSE);
		chkStatus.enable := FALSE;
		ac_setStateAfterPB;

	CTRL_AUTO_BEFORE:
		IF BetrCtrl.value = CONST.MACHINEMODES.AUTOMATIC THEN
		BetrStatus(set := TRUE, value := CONST.MACHINEMODES.AUTOMATIC);
			(*clamp.init(clk := clk);*)
			err(reset := TRUE);
			chkStatus.enable := TRUE;
			busy := FALSE;
			state := ST_IDLE;
			StateCtrl := CTRL_AUTO;
		ELSIF BetrCtrl.value = CONST.MACHINEMODES.EMERGENCYSTOP THEN
			StateCtrl := CTRL_EMERGENCYSTOP_BEFORE;
		ELSIF BetrCtrl.value = CONST.MACHINEMODES.SAFETYSTOP THEN
			StateCtrl := CTRL_SAFETYSTOP_BEFORE;
		ELSIF BetrCtrl.value = CONST.MACHINEMODES.MANUAL THEN
			StateCtrl := CTRL_MANUAL_BEFORE;
		END_IF

	(* ******************************** *)
	(* *********** AUTO *************** *)
	(* ******************************** *)
	CTRL_AUTO:
		IF BetrCtrl.value <> CONST.MACHINEMODES.AUTOMATIC THEN
			err(reset := TRUE);
			busy := TRUE;
			StateCtrl := CTRL_AUTO_AFTER;
		ELSE
			;(*ac_automatic();*)
		END_IF

	CTRL_AUTO_AFTER:
		chkStatus.enable := FALSE;
		state := ST_IDLE;
		ac_setStateAfterPB;

	CTRL_STOP_BEFORE:
		IF BetrCtrl.value = CONST.MACHINEMODES.EMERGENCYSTOP THEN
			StateCtrl := CTRL_EMERGENCYSTOP_BEFORE;
		ELSIF BetrCtrl.value = CONST.MACHINEMODES.SAFETYSTOP THEN
			StateCtrl := CTRL_SAFETYSTOP_BEFORE;
		ELSE
			state := ST_IDLE;
			StateCtrl := CTRL_STOP;
		END_IF

	CTRL_STOP:
		IF BetrCtrl.value = CONST.MACHINEMODES.EMERGENCYSTOP THEN
			StateCtrl := CTRL_EMERGENCYSTOP_BEFORE;
		ELSIF BetrCtrl.value = CONST.MACHINEMODES.SAFETYSTOP THEN
			StateCtrl := CTRL_SAFETYSTOP_BEFORE;
		ELSE
			CASE state OF
			ST_IDLE:
				state := ST_QUIT;

			ST_QUIT:
				state := ST_IDLE;
				StateCtrl := CTRL_STOP_AFTER;
			END_CASE
		END_IF

	CTRL_STOP_AFTER:
		IF BetrCtrl.value = CONST.MACHINEMODES.EMERGENCYSTOP THEN
			StateCtrl := CTRL_EMERGENCYSTOP_BEFORE;
		ELSIF BetrCtrl.value = CONST.MACHINEMODES.SAFETYSTOP THEN
			StateCtrl := CTRL_SAFETYSTOP_BEFORE;
		ELSIF BetrCtrl.value = CONST.MACHINEMODES.MANUAL THEN
			StateCtrl := CTRL_MANUAL_BEFORE;
		ELSIF BetrCtrl.value = CONST.MACHINEMODES.AUTOMATIC THEN
			StateCtrl := CTRL_AUTO_BEFORE;
		END_IF

	CTRL_RESET_START:
		BetrStatus(set := TRUE,value := CONST.MACHINEMODES.RESET);
		IF BetrCtrl.value = CONST.MACHINEMODES.EMERGENCYSTOP THEN
			StateCtrl := CTRL_EMERGENCYSTOP_BEFORE;
		ELSIF BetrCtrl.value = CONST.MACHINEMODES.SAFETYSTOP THEN
			StateCtrl := CTRL_SAFETYSTOP_BEFORE;
		ELSE
			IF axis.ctrl.busy OR axis.ctrl.cmd <> CONST.AXIS.NOACTION THEN
				axis.ctrl(cmd := CONST.AXIS.NOACTION);
			ELSE
				axis.ctrl(cmd := CONST.AXIS.RESET);
				StateCtrl := CTRL_RESET;
			END_IF
		END_IF

	CTRL_RESET:
		axis.ctrl();
		(*axis.ctrl(cmd := CONST.AXIS.RESET);**********************)
		IF BetrCtrl.value = CONST.MACHINEMODES.EMERGENCYSTOP THEN
			StateCtrl := CTRL_EMERGENCYSTOP_BEFORE;
		ELSIF BetrCtrl.value = CONST.MACHINEMODES.SAFETYSTOP THEN
			StateCtrl := CTRL_SAFETYSTOP_BEFORE;
		ELSE	manualFirst := FALSE;
			(*IF NOT axis.ctrl.busy AND axis.ctrl.MC_ReadStatus_0.Disabled THEN*)
				axis.ctrl(cmd := CONST.AXIS.POWER_OFF);(*25.06.14war NOACTION*)
			(*	axis.ctrl(cmd := CONST.AXIS.POWER_ON);(******************************)
				StateCtrl := CTRL_RESET_AFTER;
			(*END_IF*)
		END_IF

	CTRL_RESET_AFTER:
		IF BetrCtrl.value = CONST.MACHINEMODES.RESET THEN
			busy := FALSE;
		ELSE
			busy := TRUE;
		(*	clamp.init(clk := clk);*)
			err(reset := TRUE);
			IF BetrCtrl.value = CONST.MACHINEMODES.EMERGENCYSTOP THEN
				StateCtrl := CTRL_EMERGENCYSTOP_BEFORE;
			ELSIF BetrCtrl.value = CONST.MACHINEMODES.SAFETYSTOP THEN
				StateCtrl := CTRL_SAFETYSTOP_BEFORE;
			ELSIF BetrCtrl.value = CONST.MACHINEMODES.SAFETYSTOP THEN
				StateCtrl := CTRL_SAFETYSTOP_BEFORE;
			ELSIF BetrCtrl.value = CONST.MACHINEMODES.MANUAL AND safety.valid THEN
				supplydelay(IN:= TRUE, PT := T#8s);
				IF supplydelay.Q THEN
					axis.ctrl(cmd := CONST.AXIS.POWER_ON);
					busy := TRUE;
					supplydelay(IN:= FALSE);
					StateCtrl := CTRL_MANUAL_BEFORE;
				END_IF
			ELSIF BetrCtrl.value = CONST.MACHINEMODES.AUTOMATIC AND safety.valid THEN
				supplydelay(IN:= TRUE, PT := T#8s);
				IF supplydelay.Q THEN
					axis.ctrl(cmd := CONST.AXIS.POWER_ON);
					busy := TRUE;
					supplydelay(IN:= FALSE);
					StateCtrl := CTRL_AUTO_BEFORE;
				END_IF
			END_IF
		END_IF

	CTRL_SAFETYSTOP_BEFORE:
		status.isCoupled := FALSE;
		status.ready := FALSE;
		IF BetrCtrl.value = CONST.MACHINEMODES.EMERGENCYSTOP THEN
			StateCtrl := CTRL_EMERGENCYSTOP_BEFORE;
		ELSE
			BetrStatus(set := TRUE,value := CONST.MACHINEMODES.SAFETYSTOP);
			state := ST_IDLE;
			manualFirst := FALSE;
			axis.ctrl.verzoegerung	:= CONST.AXIS.EMERGENCY_DECELERATION;
			axis.ctrl.cmd := CONST.AXIS.STOP;
		(*	axis.cplOn(Execute := FALSE);*)
			StateCtrl := CTRL_SAFETYSTOP;
		END_IF

	CTRL_SAFETYSTOP:

		IF BetrCtrl.value = CONST.MACHINEMODES.EMERGENCYSTOP THEN
			StateCtrl := CTRL_EMERGENCYSTOP_BEFORE;
		ELSE
		BetrStatus(set := TRUE,value := CONST.MACHINEMODES.SAFETYSTOP);
			IF axis.ctrl.MC_ReadStatus_0.StandStill THEN
				axis.ctrl.cmd := CONST.AXIS.POWER_OFF;
			ELSIF axis.ctrl.MC_ReadStatus_0.Disabled THEN
				axis.ctrl.cmd := CONST.AXIS.NOACTION;
				StateCtrl := CTRL_SAFETYSTOP_AFTER;
			END_IF
		END_IF

	CTRL_SAFETYSTOP_AFTER:
		busy := FALSE;
		manualFirst := FALSE;
					status.ready := FALSE;
		IF BetrCtrl.value = CONST.MACHINEMODES.EMERGENCYSTOP THEN
			busy := TRUE;
			StateCtrl := CTRL_EMERGENCYSTOP_BEFORE;
		ELSIF BetrCtrl.value = CONST.MACHINEMODES.MANUAL AND safety.valid THEN
				IF axis.ctrl.MC_ReadStatus_0.Errorstop THEN
					axis.ctrl(cmd := CONST.AXIS.RESET);
				END_IF
				supplydelay(IN:= TRUE, PT := T#8s);
				IF supplydelay.Q THEN
					axis.ctrl(cmd := CONST.AXIS.POWER_ON);
					busy := TRUE;
					supplydelay(IN:= FALSE);
					StateCtrl := CTRL_MANUAL_BEFORE;
				END_IF
		ELSIF BetrCtrl.value = CONST.MACHINEMODES.AUTOMATIC AND safety.valid THEN
				IF axis.ctrl.MC_ReadStatus_0.Errorstop THEN
					axis.ctrl(cmd := CONST.AXIS.RESET);
				END_IF
				supplydelay(IN:= TRUE, PT := T#8s);
				IF supplydelay.Q THEN
					axis.ctrl(cmd := CONST.AXIS.POWER_ON);
					busy := TRUE;
					supplydelay(IN:= FALSE);
					StateCtrl := CTRL_AUTO_BEFORE;
				END_IF

		END_IF

	CTRL_EMERGENCYSTOP_BEFORE:
//		status.isCoupled := FALSE;
//		status.ready := FALSE;
//		manualFirst := FALSE;
//		axis.ctrl(cmd := CONST.AXIS.POWER_OFF);(*drvCtrl.resetRelease(ref := axis.ctrl.ref);*)
//		BetrStatus(set := TRUE, value := CONST.MACHINEMODES.EMERGENCYSTOP);
//		busy := FALSE;
		//		StateCtrl := CTRL_EMERGENCYSTOP;
		BetrStatus(set := TRUE, value := CONST.MACHINEMODES.EMERGENCYSTOP);
		status.isCoupled := FALSE;
		status.ready := FALSE;
		manualFirst := FALSE;
		IF  axis.ctrl.MC_ReadStatus_0.ContinuousMotion OR axis.ctrl.MC_ReadStatus_0.DiscreteMotion
			OR axis.ctrl.MC_ReadStatus_0.SynchronizedMotion THEN //alle Zustände in denen die Achse sich bewegen kann
			axis.ctrl.verzoegerung:= CONST.AXIS.EMERGENCY_DECELERATION; (*200m/min in 3 sek*); (* von 200m/min in 2 sek*)
			axis.ctrl.cmd := CONST.AXIS.STOP;
			state := ST_IDLE;
			StateCtrl := CTRL_EMERGENCYSTOP;
		ELSE //wenn die Maschine eingeschaltet wird
			axis.ctrl.cmd := CONST.AXIS.NOACTION;
			state := ST_IDLE;
			StateCtrl := CTRL_EMERGENCYSTOP;
		END_IF

	CTRL_EMERGENCYSTOP:
		status.isCoupled := FALSE;
		status.ready := FALSE;
			IF BetrCtrl.value = CONST.MACHINEMODES.EMERGENCYSTOP THEN
				IF axis.ctrl.MC_ReadStatus_0.StandStill THEN
					axis.ctrl.cmd := CONST.AXIS.POWER_OFF;
					busy := FALSE;
				ELSIF axis.ctrl.MC_ReadStatus_0.Disabled THEN
					axis.ctrl.cmd := CONST.AXIS.NOACTION;
					busy := FALSE;
				END_IF
			ELSE
				busy := TRUE;
				timer(IN := TRUE, PT := T#2s);
				StateCtrl := CTRL_EMERGENCYSTOP_AFTER;
			END_IF

	CTRL_EMERGENCYSTOP_AFTER:
		timer();
		IF BetrCtrl.value = CONST.MACHINEMODES.EMERGENCYSTOP THEN
			timer(IN := FALSE);
			BetrStatus(set := TRUE , value := CONST.MACHINEMODES.EMERGENCYSTOP);
			busy := FALSE;
			StateCtrl := CTRL_EMERGENCYSTOP;
		ELSIF timer.Q THEN
			timer(IN := FALSE);
			StateCtrl := CTRL_RESET_START;
		END_IF

	ELSE
		;
	END_CASE
//	axis.ctrl.BasicControl.Parameter.Deceleration	:= 40000.0; //only for initialization
//	axis.ctrl.BasicControl.Parameter.Acceleration	:= 40000.0;

END_FUNCTION_BLOCK
```

#### ac_manualPB.st
```iecst
(********************************************************************
 * COPYRIGHT -- Microsoft
 ********************************************************************
 * Programm: MAIN
 * Datei: ac_manualPB.st
 * Autor: Awalz
 * Erstellt: 7. Mai 2014
 ********************************************************************
 * Implementierung des Programms MAIN
 ********************************************************************)

 (*<$Description$> Fügt eine neue Aktion zum IEC Programm oder Bibliothek </$Description$>*)
ACTION ac_manualPB:
//	axis.ctrl();
	config( machineMasterCtrl := machineMaster, axis := axis, status := status);
	CASE state OF
	ST_IDLE:
//		IF config.busy OR config.cmd <> CONST.CUTTINGUNIT.CMDs.NO_CMD THEN
//			config(cmd := CONST.CUTTINGUNIT.CMDs.NO_CMD, machineMasterCtrl := machineMaster, axis := axis, status := status);
		IF manualFirst  OR mode <> status.mode (*OR NewData *)THEN
			IF NOT status.isCoupled AND mode = CONST.UNITMODEs.ENABLE THEN
				config(cmd := CONST.CUTTINGUNIT.CMDs.CPL_ON, machineMasterCtrl := machineMaster, axis := axis, status := status);
				state := ST_CPL_WAIT;
			ELSIF mode <> CONST.UNITMODEs.ENABLE AND status.isCoupled THEN
				config(cmd := CONST.CUTTINGUNIT.CMDs.CPL_OFF, machineMasterCtrl := machineMaster, axis := axis, status := status);
				state := ST_CPL_WAIT;
			ELSE
				NewData := FALSE;
				manualFirst := FALSE;
			END_IF
///////////////////////////////////////////////////
//			ELSIF cmdCtrl.value = CONST.CUTTINGUNIT.CMDs.MOVEFW OR cmdCtrl.value = CONST.CUTTINGUNIT.CMDs.MOVEBW THEN
//					state := 	ST_MOVE_START;
//////////////////////////////
		ELSIF cmdCtrl.value <> CONST.CUTTINGUNIT.CMDs.NO_CMD THEN
			cmdStatus(set := TRUE, value := cmdCtrl.value);
			busy := TRUE;
			state := ST_FUNCTION_START;
		END_IF

	ST_CPL_WAIT:
		config( machineMasterCtrl := machineMaster, axis := axis, status := status);
		IF NOT config.busy THEN
			IF config.err.flag THEN
				err := config.err;
				err.state := state;
				state := ST_ERROR;
			ELSE
				manualFirst := FALSE;
				state := ST_IDLE;
			END_IF
			config(cmd := CONST.CUTTINGUNIT.CMDs.NO_CMD, machineMasterCtrl := machineMaster, axis := axis, status := status );
		END_IF

	ST_FUNCTION_START:
//		IF config.busy (*OR config.cmd <> CONST.CUTTINGUNIT.CMDs.NO_CMD*) THEN
//			config(cmd := CONST.CUTTINGUNIT.CMDs.NO_CMD, machineMasterCtrl := machineMaster, axis := axis, status := status);
//		ELSE
			config(cmd := cmdStatus.value, machineMasterCtrl := machineMaster, axis := axis, status := status);
			state := ST_FUNCTION;
	(*	END_IF*)

	ST_FUNCTION:
////		config( machineMasterCtrl := machineMaster, axis := axis, status := status);
////		IF NOT config.busy THEN
////			IF config.err.flag THEN
////				err := config.err;
////				err.state := state;
////			END_IF
////		config(cmd := CONST.CUTTINGUNIT.CMDs.NO_CMD, machineMasterCtrl := machineMaster, axis := axis, status := status );
////			state := ST_FUNCTION_QUIT;
		IF cmdCtrl.value = CONST.CUTTINGUNIT.CMDs.NO_CMD THEN
			config(cmd := CONST.CUTTINGUNIT.CMDs.NO_CMD, machineMasterCtrl := machineMaster, axis := axis, status := status );
			state := ST_FUNCTION_QUIT;
		END_IF

	ST_FUNCTION_QUIT:
		busy := FALSE;
		IF cmdCtrl.value = CONST.CUTTINGUNIT.CMDs.NO_CMD THEN
			cmdStatus(set :=TRUE, value := CONST.CUTTINGUNIT.CMDs.NO_CMD);
			state := ST_IDLE;
		END_IF

	ST_ERROR:
		err.flag := TRUE;
		busy := FALSE;
		IF BetrCtrl.value <> CONST.MACHINEMODES.MANUAL THEN
			state := ST_IDLE;
			err(reset := TRUE);
			busy := TRUE;
			StateCtrl := CTRL_MANUAL_AFTER;
		END_IF
	END_CASE

END_ACTION
```

#### FB_PULLBRAEKUNIT.st
```iecst
(********************************************************************
 * COPYRIGHT -- Microsoft
 ********************************************************************
 * Programm: MAIN
 * Datei: FB_PULLBRAEKUNIT.st
 * Autor: Awalz
 * Erstellt: 27. März 2014
 ********************************************************************
 * Implementierung des Programms MAIN
 ********************************************************************)

(*<$Description$> TODO: Bitte Kommentar hier einzufügen </$Description$>*)
FUNCTION_BLOCK FB_PULLBREAKUNIT
END_FUNCTION_BLOCK
```

#### FB_PULLBREAK_AXIS.st
```iecst
(********************************************************************
 * COPYRIGHT -- Microsoft
 ********************************************************************
 * Programm: MAIN
 * Datei: FB_PULLBREAK_AXIS.st
 * Autor: Awalz
 * Erstellt: 7. Mai 2014
 ********************************************************************
 * Implementierung des Programms MAIN
 ********************************************************************)

 (*<$Description$> TODO: Bitte Kommentar hier einzufügen </$Description$>*)
FUNCTION_BLOCK FB_PULLBREAK_AXIS
END_FUNCTION_BLOCK
```

#### Package Logical/MainMachineCtrl/MAIN/TurnGrindwinderUnit - Neues leeres Paket

#### FB_TurnGridUnitCtrl.st
```iecst
(********************************************************************
 * COPYRIGHT -- Microsoft
 ********************************************************************
 * Programm: MAIN
 * Datei: FB_TurnGridUnitCtrl.st
 * Autor: awalz
 * Erstellt: 25. Juni 2014
 ********************************************************************
 * Implementierung des Programms MAIN
 ********************************************************************)

(* TODO: Bitte Kommentar hier einfügen *)
FUNCTION_BLOCK FB_TurnGridUnitCtrl
	gridwinderright.ctrl(BetrCtrl := BetrCtrl, machineaxis := machineaxis, axis := gridwinderright.axis,
					 status := gridwinderright.status, data := gridwinderright.data);
	gridwinderleft.ctrl(BetrCtrl := BetrCtrl, machineaxis := machineaxis, axis := gridwinderleft.axis,
					 status := gridwinderleft.status,  data := gridwinderleft.data);
	refSwitchConfig(Enable := TRUE); // OKrebs // 13.04.17
	SwitchConfig.refSwitchChannelName := ADR('DigitalInput08');
	SwitchConfig.refSwitchDeviceName := ADR('SL1.IF1.ST16.IF1.ST6');
	SwitchConfig.Execute := TRUE;
	SwitchConfig();
	feeder();
	feederstatus(axisState := feeder.MC_ReadStatus_0);
	TurnGrWinKeysbox(clk := clk);
//	ac_manualTurnGrd; (*Aufruf der Action*) // OKrebs 26.04.17
 	IF feeder.MC_ReadActualPosition_0.Position > 170000 AND feeder.MC_ReadActualPosition_0.Position < 190000 AND feeder.MC_ReadStatus_0.DiscreteMotion  THEN
				gridwinderright.data.recipeData.mode := CONST.UNITMODEs.AXIS_OFF;
				gridwinderleft.data.recipeData.mode := CONST.UNITMODEs.ENABLE;
	ELSIF (feeder.MC_ReadActualPosition_0.Position > 350000 OR feeder.MC_ReadActualPosition_0.Position < 10000) AND feeder.MC_ReadStatus_0.DiscreteMotion  THEN
				gridwinderright.data.recipeData.mode := CONST.UNITMODEs.ENABLE;
				gridwinderleft.data.recipeData.mode := CONST.UNITMODEs.AXIS_OFF;
	ELSE

 	END_IF

 	IF TurnGrWinKeysbox.GridWinleftkey.buttonDown.LDT.button AND TurnGrWinKeysbox.GridWinleftkey.buttonDown.LDT.button AND feeder.MC_ReadStatus_0.Disabled THEN
		feeder.cmd := CONST.AXIS.POWER_ON;
	ELSIF TurnGrWinKeysbox.GridWinleftkey.buttonDown.LDT.button AND TurnGrWinKeysbox.GridWinleftkey.buttonDown.LDT.button AND feeder.MC_ReadStatus_0.Errorstop THEN
		feeder.cmd := CONST.AXIS.RESET;
	END_IF
	IF feeder.MC_ReadStatus_0.StandStill THEN
		TurnGrWinKeysbox.feederturnkey.LDT.aktion := CONST.LAMP.ON;
	ELSIF feeder.MC_ReadStatus_0.Disabled THEN
		TurnGrWinKeysbox.feederturnkey.LDT.aktion := CONST.LAMP.BLINK1000;
	ELSIF feeder.MC_ReadStatus_0.Errorstop THEN
		TurnGrWinKeysbox.feederturnkey.LDT.aktion := CONST.LAMP.BLINK200;
	END_IF
//	IF NOT feeder.MC_ReadStatus_0.Disabled THEN
//		IF TurnGrWinKeysbox.feederturnkey.LDT.rtrig.Q THEN
//			 feeder(cmd :=  CONST.AXIS.JOG_POS, velocity := 0.024);
//			axisstep := ST_STOP;
//		ELSE

//	IF gridwinderright.data.recipeData.mode = CONST.UNITMODEs.ENABLE THEN
	R_TRIG_feederturnkey.CLK := TurnGrWinKeysbox.feederturnkey.LDT.button;
	R_TRIG_feederturnkey();

	CASE axisstep OF

		ST_IDLE:
			IF NOT feeder.BasicControl.AxisState.Homed AND feeder.MC_ReadStatus_0.StandStill THEN // OKrebs // 13.04.17
				IF FeederHomeButton THEN
					feeder.BasicControl.Parameter.HomeMode := mcHOME_ABS_SWITCH;
					feeder.BasicControl.Parameter.HomePosition := 0.0;
					feeder(cmd := CONST.AXIS.CALIBR);
				END_IF
			ELSIF NOT panel.LDTStop.LDT.button THEN
				FeederHomeButton := FALSE;
				axisstep := ST_STOP;
			ELSIF feeder.BasicControl.AxisState.Homed AND NOT feeder.MC_ReadStatus_0.Disabled AND NOT feeder.MC_ReadStatus_0.Homing THEN // OKrebs // 13.04.17
				IF R_TRIG_feederturnkey.Q OR test THEN
					IF  (feeder.MC_ReadActualPosition_0.Position < 179000) OR (feeder.MC_ReadActualPosition_0.Position > 359000) THEN
						feeder(cmd :=  CONST.AXIS.SETPOS, velocity := 1.8, position := 180000);  (*Position aus Rezept*)(*5U/min/60s *360000*16666*)
						merker := TRUE;
					ELSE
						feeder(cmd :=  CONST.AXIS.SETPOS, velocity := 1.8, position := 0);  (*Position aus Rezept*)(*5U/min/60s *360000*16666*)
						merker := TRUE;
					END_IF
				ELSIF NOT TurnGrWinKeysbox.feederturnkey.LDT.button AND merker AND NOT test THEN
					axisstep := ST_STOP;
				END_IF
			END_IF // OKrebs // 13.04.17
		ST_STOP:
			feeder(cmd := CONST.AXIS.STOP, verzoegerung := feeder.BasicControl.Parameter.Deceleration);
			merker := FALSE;
			axisstep := ST_NOACTION;

		ST_NOACTION:
         	feeder(cmd := CONST.AXIS.NOACTION);
		 	axisstep := ST_IDLE;
	END_CASE

CASE StateCtrl OF
		CTRL_FIRST_START:
		busy := TRUE;
		StateCtrl := CTRL_EMERGENCYSTOP_BEFORE;

	CTRL_MANUAL_BEFORE:
		IF BetrCtrl.value = CONST.MACHINEMODES.MANUAL THEN
			gridwinderright.ctrl.BetrCtrl(set := TRUE,value := CONST.MACHINEMODES.MANUAL);
			gridwinderleft.ctrl.BetrCtrl(set := TRUE,value := CONST.MACHINEMODES.MANUAL);
			IF NOT gridwinderright.ctrl.busy AND NOT gridwinderleft.ctrl.busy THEN
				BetrStatus(set := TRUE, value := BetrCtrl.value);
				busy := FALSE;
				err(reset := TRUE);
				state := ST_IDLE;
				StateCtrl := CTRL_MANUAL;
			END_IF
		ELSIF BetrCtrl.value = CONST.MACHINEMODES.EMERGENCYSTOP THEN
			StateCtrl := CTRL_EMERGENCYSTOP_BEFORE;
		ELSIF BetrCtrl.value = CONST.MACHINEMODES.SAFETYSTOP THEN
			StateCtrl := CTRL_SAFETYSTOP_BEFORE;
		ELSIF BetrCtrl.value = CONST.MACHINEMODES.AUTOMATIC THEN
			StateCtrl := CTRL_AUTO_BEFORE;
		END_IF

	CTRL_MANUAL://11
		IF BetrCtrl.value <> CONST.MACHINEMODES.MANUAL THEN
			err(reset := TRUE);
			busy := TRUE;
			StateCtrl := CTRL_MANUAL_AFTER;
		ELSE
		(*	ac_manualTurnGrd; (*Aufruf der Action*)
		END_IF

	CTRL_MANUAL_AFTER://12
		(*chkStatus.enable := FALSE;*)
		ac_setStateAfterUnwinder; (*Aufruf der Action*)

	CTRL_AUTO_BEFORE://20
		IF BetrCtrl.value = CONST.MACHINEMODES.AUTOMATIC THEN
			BetrStatus(set := TRUE, value := CONST.MACHINEMODES.AUTOMATIC);
			(*clamp.init(clk := clk);
			chkStatus.enable := TRUE;*)
			err(reset := TRUE);
			busy := FALSE;
			state := ST_IDLE;
			StateCtrl := CTRL_AUTO;
		ELSIF BetrCtrl.value = CONST.MACHINEMODES.EMERGENCYSTOP THEN
			StateCtrl := CTRL_EMERGENCYSTOP_BEFORE;
		ELSIF BetrCtrl.value = CONST.MACHINEMODES.SAFETYSTOP THEN
			StateCtrl := CTRL_SAFETYSTOP_BEFORE;
		ELSIF BetrCtrl.value = CONST.MACHINEMODES.MANUAL THEN
			StateCtrl := CTRL_MANUAL_BEFORE;
		END_IF

	(* ******************************** *)
	(* *********** AUTO *************** *)
	(* ******************************** *)
	CTRL_AUTO://22
		IF BetrCtrl.value <> CONST.MACHINEMODES.AUTOMATIC THEN
			err(reset := TRUE);
			busy := TRUE;
			StateCtrl := CTRL_AUTO_AFTER;
		ELSE
			(*ac_automatic();*)
		END_IF

	CTRL_AUTO_AFTER://23
		(*chkStatus.enable := FALSE;*)
		state := ST_IDLE;
		ac_setStateAfterUnwinder;

	CTRL_STOP_BEFORE://50
		IF BetrCtrl.value = CONST.MACHINEMODES.EMERGENCYSTOP THEN
			StateCtrl := CTRL_EMERGENCYSTOP_BEFORE;
		ELSIF BetrCtrl.value = CONST.MACHINEMODES.SAFETYSTOP THEN
			StateCtrl := CTRL_SAFETYSTOP_BEFORE;
		ELSE
			state := ST_IDLE;
			StateCtrl := CTRL_STOP;
		END_IF

	CTRL_STOP:
		IF BetrCtrl.value = CONST.MACHINEMODES.EMERGENCYSTOP THEN
			StateCtrl := CTRL_EMERGENCYSTOP_BEFORE;
		ELSIF BetrCtrl.value = CONST.MACHINEMODES.SAFETYSTOP THEN
			StateCtrl := CTRL_SAFETYSTOP_BEFORE;
		ELSE
			CASE state OF
			ST_IDLE:
				state := ST_QUIT;

			ST_QUIT:
				state := ST_IDLE;
				StateCtrl := CTRL_STOP_AFTER;
			END_CASE
		END_IF

	CTRL_STOP_AFTER:
		IF BetrCtrl.value = CONST.MACHINEMODES.EMERGENCYSTOP THEN
			StateCtrl := CTRL_EMERGENCYSTOP_BEFORE;
		ELSIF BetrCtrl.value = CONST.MACHINEMODES.SAFETYSTOP THEN
			StateCtrl := CTRL_SAFETYSTOP_BEFORE;
		ELSIF BetrCtrl.value = CONST.MACHINEMODES.MANUAL THEN
			StateCtrl := CTRL_MANUAL_BEFORE;
		ELSIF BetrCtrl.value = CONST.MACHINEMODES.AUTOMATIC THEN
			StateCtrl := CTRL_AUTO_BEFORE;
		END_IF

	CTRL_RESET_START:
		BetrStatus(set := TRUE, value := CONST.MACHINEMODES.RESET);
		IF BetrCtrl.value = CONST.MACHINEMODES.EMERGENCYSTOP THEN
			StateCtrl := CTRL_EMERGENCYSTOP_BEFORE;
		ELSIF BetrCtrl.value = CONST.MACHINEMODES.SAFETYSTOP THEN
			StateCtrl := CTRL_SAFETYSTOP_BEFORE;
		ELSE
			IF feeder.busy OR feeder.cmd <> CONST.AXIS.NOACTION THEN
				feeder(cmd := CONST.AXIS.NOACTION);
			ELSE
				feeder.cmd := CONST.AXIS.RESET;
				StateCtrl := CTRL_RESET;
			END_IF
		END_IF

	CTRL_RESET:

		IF BetrCtrl.value = CONST.MACHINEMODES.EMERGENCYSTOP THEN
			StateCtrl := CTRL_EMERGENCYSTOP_BEFORE;
		ELSIF BetrCtrl.value = CONST.MACHINEMODES.SAFETYSTOP THEN
			StateCtrl := CTRL_SAFETYSTOP_BEFORE;
		ELSE
			(*IF NOT feeder.busy THEN*)
				feeder.cmd := CONST.AXIS.NOACTION;
				StateCtrl := CTRL_RESET_AFTER;
		(*	END_IF*)
		END_IF

	CTRL_RESET_AFTER:
		IF BetrCtrl.value = CONST.MACHINEMODES.RESET THEN
			busy := FALSE;
		ELSE
			busy := TRUE;
			(*clamp.init(clk := clk);
			err.reset();*)
			err(reset := TRUE);
			IF BetrCtrl.value = CONST.MACHINEMODES.EMERGENCYSTOP THEN
				StateCtrl := CTRL_EMERGENCYSTOP_BEFORE;
			ELSIF BetrCtrl.value = CONST.MACHINEMODES.SAFETYSTOP THEN
				StateCtrl := CTRL_SAFETYSTOP_BEFORE;
			ELSIF BetrCtrl.value = CONST.MACHINEMODES.SAFETYSTOP THEN
				StateCtrl := CTRL_SAFETYSTOP_BEFORE;
			ELSIF BetrCtrl.value = CONST.MACHINEMODES.MANUAL THEN
					supplydelay(IN:= TRUE, PT := T#8s);
				IF supplydelay.Q THEN
					feeder(cmd := CONST.AXIS.POWER_ON);
					busy := TRUE;
					supplydelay(IN:= FALSE);
					StateCtrl := CTRL_MANUAL_BEFORE;
				END_IF
			ELSIF BetrCtrl.value = CONST.MACHINEMODES.AUTOMATIC THEN
				supplydelay(IN:= TRUE, PT := T#8s);
				IF supplydelay.Q THEN
					feeder(cmd := CONST.AXIS.POWER_ON);
					busy := TRUE;
					supplydelay(IN:= FALSE);
					StateCtrl := CTRL_AUTO_BEFORE;
				END_IF
			END_IF
		END_IF

	CTRL_SAFETYSTOP_BEFORE://82
		IF BetrCtrl.value = CONST.MACHINEMODES.EMERGENCYSTOP THEN
			StateCtrl := CTRL_EMERGENCYSTOP_BEFORE;
		ELSE
			feeder.verzoegerung	:= CONST.AXIS.EMERGENCY_DECELERATION;
			feeder.cmd := CONST.AXIS.STOP;//24.03.15
			BetrStatus.set := TRUE;
			BetrStatus.value := CONST.MACHINEMODES.SAFETYSTOP;
			state := ST_IDLE;
			StateCtrl := CTRL_SAFETYSTOP;
		END_IF

	CTRL_SAFETYSTOP://85
		IF BetrCtrl.value = CONST.MACHINEMODES.EMERGENCYSTOP THEN
			StateCtrl := CTRL_EMERGENCYSTOP_BEFORE;
		ELSE
		BetrStatus(set := TRUE, value := CONST.MACHINEMODES.SAFETYSTOP);
			IF feeder.MC_ReadStatus_0.StandStill THEN //24.03.15
				feeder.cmd := CONST.AXIS.POWER_OFF;
			ELSIF feeder.MC_ReadStatus_0.Disabled THEN
				feeder.cmd := CONST.AXIS.NOACTION;
				StateCtrl := CTRL_SAFETYSTOP_AFTER;
			END_IF
//			CASE state OF
//			ST_IDLE:
//				IF NOT gridwinderright.ctrl.busy AND NOT gridwinderleft.ctrl.busy THEN
//					state := ST_QUIT;
//				END_IF
//			ST_QUIT:
//				state := ST_IDLE;
//				BetrStatus(set := TRUE, value := CONST.MACHINEMODES.SAFETYSTOP);
//				StateCtrl := CTRL_SAFETYSTOP_AFTER;
//			END_CASE
		END_IF

	CTRL_SAFETYSTOP_AFTER:
		busy := FALSE;
		IF BetrCtrl.value = CONST.MACHINEMODES.EMERGENCYSTOP THEN
			busy := TRUE;
			StateCtrl := CTRL_EMERGENCYSTOP_BEFORE;
		ELSIF BetrCtrl.value = CONST.MACHINEMODES.MANUAL THEN
				supplydelay(IN:= TRUE, PT := T#8s);
				IF supplydelay.Q THEN
					feeder(cmd := CONST.AXIS.POWER_ON);
					busy := TRUE;
					supplydelay(IN:= FALSE);
					StateCtrl := CTRL_MANUAL_BEFORE;
				END_IF
		ELSIF BetrCtrl.value = CONST.MACHINEMODES.AUTOMATIC THEN
				supplydelay(IN:= TRUE, PT := T#8s);
				IF supplydelay.Q THEN
					feeder(cmd := CONST.AXIS.POWER_ON);
					busy := TRUE;
					supplydelay(IN:= FALSE);
					feeder(cmd := CONST.AXIS.POWER_ON);
					StateCtrl := CTRL_AUTO_BEFORE;
				END_IF
		END_IF

	CTRL_EMERGENCYSTOP_BEFORE:
		gridwinderleft.ctrl.BetrCtrl(set := TRUE,value := CONST.MACHINEMODES.EMERGENCYSTOP);
		gridwinderright.ctrl.BetrCtrl(set := TRUE,value := CONST.MACHINEMODES.EMERGENCYSTOP);
			(*feeder.cmd := CONST.AXIS.POWER_OFF;*)//24.03.15
		feeder.verzoegerung	:= CONST.AXIS.EMERGENCY_DECELERATION;//24.03.15
		feeder.cmd := CONST.AXIS.STOP;
		IF NOT gridwinderright.ctrl.busy AND NOT gridwinderright.ctrl.busy THEN

			IF gridwinderright.ctrl.BetrStatus.value = CONST.MACHINEMODES.EMERGENCYSTOP
				AND gridwinderleft.ctrl.BetrStatus.value = CONST.MACHINEMODES.EMERGENCYSTOP THEN
				BetrStatus(set := TRUE, value := CONST.MACHINEMODES.EMERGENCYSTOP);
				StateCtrl := CTRL_EMERGENCYSTOP;
			END_IF

		END_IF

	CTRL_EMERGENCYSTOP:

		IF BetrCtrl.value = CONST.MACHINEMODES.EMERGENCYSTOP THEN
			IF feeder.MC_ReadStatus_0.StandStill THEN
				feeder.cmd := CONST.AXIS.POWER_OFF;
				busy := FALSE;
			ELSIF feeder.MC_ReadStatus_0.Disabled THEN
				feeder.cmd := CONST.AXIS.NOACTION;
				busy := FALSE;
			END_IF
		ELSE
			busy := TRUE;
			StateCtrl:= CTRL_RESET_START;
		END_IF

	END_CASE
	feeder.BasicControl.Parameter.Deceleration	:= 59000.0; //only for initialization
	feeder.BasicControl.Parameter.Acceleration	:= 59000.0;
END_FUNCTION_BLOCK
```

#### ac_manualTurnGrd.st
```iecst
(********************************************************************
 * COPYRIGHT -- Microsoft
 ********************************************************************
 * Programm: MAIN
 * Datei: ac_manualTurnGrd.st
 * Autor: Awalz
 * Erstellt: 5. Juni 2014
 ********************************************************************
 * Implementierung des Programms MAIN
 ********************************************************************)

 (*<$Description$> Fügt eine neue Aktion zum IEC Programm oder Bibliothek </$Description$>*)
ACTION ac_manualTurnGrd:
		IF feeder.MC_ReadStatus_0.ContinuousMotion THEN
			rtig := TRUE;
		ELSE
			rtig := FALSE;
		END_IF
		feedertrig(CLK := rtig);

	CASE state OF

		ST_IDLE:
			IF feedertrig.Q  THEN
				(*feederPosTmp := feeder.BasicControl.Status.ActPosition;*)
				feederPosTmp := feeder.MC_ReadActualPosition_0.Position;
				IF gridwinderright.data.recipeData.mode = CONST.UNITMODEs.ENABLE THEN
				(*	gridwinderright.data.machData.frictionCompensation := 1;*)
					state := ST_TURN_WAIT_RIGHT;
				ELSIF gridwinderleft.data.recipeData.mode = CONST.UNITMODEs.ENABLE THEN
					(*gridwinderleft.data.machData.frictionCompensation := 1;*)
					state := ST_TURN_WAIT_LEFT;
				END_IF

			END_IF

		ST_TURN_WAIT_RIGHT:
			IF feederPosTmp + 65000 < feeder.BasicControl.Status.ActPosition AND feeder.MC_ReadStatus_0.ContinuousMotion  THEN
				gridwinderright.data.recipeData.mode := CONST.UNITMODEs.AXIS_OFF;
				gridwinderleft.data.recipeData.mode := CONST.UNITMODEs.ENABLE;
				state := ST_IDLE;
			ELSIF NOT feeder.MC_ReadStatus_0.ContinuousMotion THEN
					state := ST_IDLE;
			END_IF

		ST_TURN_WAIT_LEFT:
			IF feederPosTmp + 65000 < feeder.BasicControl.Status.ActPosition AND feeder.MC_ReadStatus_0.ContinuousMotion THEN
				gridwinderright.data.recipeData.mode := CONST.UNITMODEs.ENABLE;
				gridwinderleft.data.recipeData.mode := CONST.UNITMODEs.AXIS_OFF;
				state := ST_IDLE;
			ELSIF NOT feeder.MC_ReadStatus_0.ContinuousMotion THEN
				state := ST_IDLE;
			END_IF

		ST_NOACTION:
				;
	END_CASE
END_ACTION
```

#### FB_TurnGridWinderUnit.st
```iecst
(********************************************************************
 * COPYRIGHT -- Microsoft
 ********************************************************************
 * Programm: MAIN
 * Datei: FB_TurnGridWinder.st
 * Autor: Awalz
 * Erstellt: 5. Juni 2014
 ********************************************************************
 * Implementierung des Programms MAIN
 ********************************************************************)

 (*<$Description$> TODO: Bitte Kommentar hier einzufügen </$Description$>*)
FUNCTION_BLOCK FB_TurnGridWinderUnit
END_FUNCTION_BLOCK
```

#### Package Logical/MainMachineCtrl/MAIN/TurnGrindwinderUnit/Gridwinder - Paket

#### FB_TunrGridWinCtrl.st
```iecst
(********************************************************************
 * COPYRIGHT -- Microsoft
 ********************************************************************
 * Programm: MAIN
 * Datei: FB_TunrGridWinCtrl.st
 * Autor: Awalz
 * Erstellt: 5. Juni 2014
 ********************************************************************
 * Implementierung des Programms MAIN
 ********************************************************************)

 (*<$Description$> TODO: Bitte Kommentar hier einzufügen </$Description$>*)
FUNCTION_BLOCK FB_TunrGridWinCtrl
	axis(machineaxis := machineaxis, data := data);
	axis.startdiameter := 110; (* Anfangsdurchmesser setzten*)
	status(axisState := axis.MC_ReadStatus_0);
	(*ac_manualGridWin*);
	IF data.recipeData.mode = CONST.UNITMODEs.ENABLE THEN
		IF data.recipeData.warnDiam < axis.LCRLimit_0.out THEN
			diameterWarning := TRUE;
		ELSE
			diameterWarning := FALSE;
		END_IF
		IF data.recipeData.stopDiam < axis.LCRLimit_0.out THEN
			diameterStop := TRUE;
		ELSE
			diameterStop := FALSE;
		END_IF
//		diameterWarning := SEL ((data.recipeData.warnDiam < axis.WNCCalcDiam_0.actDiam AND axis.WNCCalcDiam_0.actDiam > 0), FALSE, TRUE);
//		diameterStop := SEL((data.recipeData.stopDiam < axis.WNCCalcDiam_0.actDiam AND axis.WNCCalcDiam_0.actDiam > 0), FALSE, TRUE);
	ELSE
		diameterStop := FALSE;
		diameterWarning := FALSE;
	END_IF
	chkStatus(setMode := data.recipeData.mode, status := status);
//	clamp(clk := clk);
	CASE StateCtrl OF
	CTRL_FIRST_START:
		busy := TRUE;
		(*axis.ctrl.BasicControl.Command.Power := TRUE;*)
		StateCtrl := CTRL_EMERGENCYSTOP_BEFORE;

	CTRL_MANUAL_BEFORE:
		IF BetrCtrl.value = CONST.MACHINEMODES.MANUAL THEN
		(*	clamp.init(clk := clk);*)
			BetrStatus(set := TRUE, value := CONST.MACHINEMODES.MANUAL);
			chkStatus.enable := TRUE;
			err(reset := TRUE);
			busy := FALSE;
			timer(IN:= FALSE);
			state := ST_IDLE;
			manualFirst := TRUE;
			StateCtrl := CTRL_MANUAL;
		ELSIF BetrCtrl.value = CONST.MACHINEMODES.EMERGENCYSTOP THEN
			StateCtrl := CTRL_EMERGENCYSTOP_BEFORE;
		ELSIF BetrCtrl.value = CONST.MACHINEMODES.SAFETYSTOP THEN
			StateCtrl := CTRL_SAFETYSTOP_BEFORE;
		ELSIF BetrCtrl.value = CONST.MACHINEMODES.AUTOMATIC THEN
			StateCtrl := CTRL_AUTO_BEFORE;
		END_IF

	CTRL_MANUAL:
		IF BetrCtrl.value <> CONST.MACHINEMODES.MANUAL THEN
			err(reset := TRUE);
			busy := TRUE;

			StateCtrl := CTRL_MANUAL_AFTER;
	(*ELSIF axis.ctrl.MC_ReadStatus_0.StandStill THEN
				timer(IN := TRUE, PT := T#8s);
				IF timer.Q THEN
					ac_manualPB;
				END_IF*)
		ELSE
			ac_manualGridWin;
		END_IF

	CTRL_MANUAL_AFTER:
		timer(IN:= FALSE);
		chkStatus.enable := FALSE;
		ac_TurnGridwinSetAfter;

	CTRL_AUTO_BEFORE:
		IF BetrCtrl.value = CONST.MACHINEMODES.AUTOMATIC THEN
		BetrStatus(set := TRUE, value := CONST.MACHINEMODES.AUTOMATIC);
			(*clamp.init(clk := clk);*)
			err(reset := TRUE);
			chkStatus.enable := TRUE;
			busy := FALSE;
			state := ST_IDLE;
			StateCtrl := CTRL_AUTO;
		ELSIF BetrCtrl.value = CONST.MACHINEMODES.EMERGENCYSTOP THEN
			StateCtrl := CTRL_EMERGENCYSTOP_BEFORE;
		ELSIF BetrCtrl.value = CONST.MACHINEMODES.SAFETYSTOP THEN
			StateCtrl := CTRL_SAFETYSTOP_BEFORE;
		ELSIF BetrCtrl.value = CONST.MACHINEMODES.MANUAL THEN
			StateCtrl := CTRL_MANUAL_BEFORE;
		END_IF

	(* ******************************** *)
	(* *********** AUTO *************** *)
	(* ******************************** *)
	CTRL_AUTO:
		IF BetrCtrl.value <> CONST.MACHINEMODES.AUTOMATIC THEN
			err(reset := TRUE);
			busy := TRUE;
			StateCtrl := CTRL_AUTO_AFTER;
		ELSE
			ac_manualGridWin;
		END_IF

	CTRL_AUTO_AFTER:
		chkStatus.enable := FALSE;
		state := ST_IDLE;
		ac_setStateAfterPB;

	CTRL_STOP_BEFORE:
		IF BetrCtrl.value = CONST.MACHINEMODES.EMERGENCYSTOP THEN
			StateCtrl := CTRL_EMERGENCYSTOP_BEFORE;
		ELSIF BetrCtrl.value = CONST.MACHINEMODES.SAFETYSTOP THEN
			StateCtrl := CTRL_SAFETYSTOP_BEFORE;
		ELSE
			state := ST_IDLE;
			StateCtrl := CTRL_STOP;
		END_IF

	CTRL_STOP:
		IF BetrCtrl.value = CONST.MACHINEMODES.EMERGENCYSTOP THEN
			StateCtrl := CTRL_EMERGENCYSTOP_BEFORE;
		ELSIF BetrCtrl.value = CONST.MACHINEMODES.SAFETYSTOP THEN
			StateCtrl := CTRL_SAFETYSTOP_BEFORE;
		ELSE
			CASE state OF
			ST_IDLE:
				state := ST_QUIT;

			ST_QUIT:
				state := ST_IDLE;
				StateCtrl := CTRL_STOP_AFTER;
			END_CASE
		END_IF

	CTRL_STOP_AFTER:
		IF BetrCtrl.value = CONST.MACHINEMODES.EMERGENCYSTOP THEN
			StateCtrl := CTRL_EMERGENCYSTOP_BEFORE;
		ELSIF BetrCtrl.value = CONST.MACHINEMODES.SAFETYSTOP THEN
			StateCtrl := CTRL_SAFETYSTOP_BEFORE;
		ELSIF BetrCtrl.value = CONST.MACHINEMODES.MANUAL THEN
			StateCtrl := CTRL_MANUAL_BEFORE;
		ELSIF BetrCtrl.value = CONST.MACHINEMODES.AUTOMATIC THEN
			StateCtrl := CTRL_AUTO_BEFORE;
		END_IF

	CTRL_RESET_START:
		BetrStatus(set := TRUE,value := CONST.MACHINEMODES.RESET);
		IF BetrCtrl.value = CONST.MACHINEMODES.EMERGENCYSTOP THEN
			StateCtrl := CTRL_EMERGENCYSTOP_BEFORE;
		ELSIF BetrCtrl.value = CONST.MACHINEMODES.SAFETYSTOP THEN
			StateCtrl := CTRL_SAFETYSTOP_BEFORE;
		ELSE;
			IF axis.busy OR  axis.cmd <> CONST.AXIS.NOACTION THEN
				axis.cmd := CONST.AXIS.NOACTION;
			ELSE
				axis.cmd := CONST.AXIS.RESET;
				StateCtrl := CTRL_RESET;
			END_IF
		END_IF

	CTRL_RESET:
	(*	axis.ctrl();*)
		(*axis.ctrl(cmd := CONST.AXIS.RESET);**********************)
		IF BetrCtrl.value = CONST.MACHINEMODES.EMERGENCYSTOP THEN
			StateCtrl := CTRL_EMERGENCYSTOP_BEFORE;
		ELSIF BetrCtrl.value = CONST.MACHINEMODES.SAFETYSTOP THEN
			StateCtrl := CTRL_SAFETYSTOP_BEFORE;
		ELSE
			IF NOT axis.busy AND axis.MC_ReadStatus_0.Disabled THEN
				axis.cmd := CONST.AXIS.NOACTION;
				StateCtrl := CTRL_RESET_AFTER;
			END_IF
		END_IF

	CTRL_RESET_AFTER:
		IF BetrCtrl.value = CONST.MACHINEMODES.RESET THEN
			busy := FALSE;
		ELSE
			busy := TRUE;
			err(reset := TRUE);
			IF BetrCtrl.value = CONST.MACHINEMODES.EMERGENCYSTOP THEN
				StateCtrl := CTRL_EMERGENCYSTOP_BEFORE;
			ELSIF BetrCtrl.value = CONST.MACHINEMODES.SAFETYSTOP THEN
				StateCtrl := CTRL_SAFETYSTOP_BEFORE;
			ELSIF BetrCtrl.value = CONST.MACHINEMODES.SAFETYSTOP THEN
				StateCtrl := CTRL_SAFETYSTOP_BEFORE;
			ELSIF BetrCtrl.value = CONST.MACHINEMODES.MANUAL THEN
				supplydelay(IN:= TRUE, PT := T#8s);
				IF supplydelay.Q THEN
					axis.cmd := CONST.AXIS.POWER_ON;
					busy := TRUE;
					supplydelay(IN:= FALSE);
					StateCtrl := CTRL_MANUAL_BEFORE;
				END_IF
			ELSIF BetrCtrl.value = CONST.MACHINEMODES.AUTOMATIC  THEN
				supplydelay(IN:= TRUE, PT := T#8s);
				IF supplydelay.Q THEN
					axis.cmd := CONST.AXIS.POWER_ON;
					busy := TRUE;
					supplydelay(IN:= FALSE);
					StateCtrl := CTRL_AUTO_BEFORE;
				END_IF
			END_IF
		END_IF

	CTRL_SAFETYSTOP_BEFORE:
		status.isCoupled := FALSE;
		status.ready := FALSE;
		IF BetrCtrl.value = CONST.MACHINEMODES.EMERGENCYSTOP THEN
			StateCtrl := CTRL_EMERGENCYSTOP_BEFORE;
		ELSE
			BetrStatus(set := TRUE,value := CONST.MACHINEMODES.SAFETYSTOP);
			state := ST_IDLE;
			axis.deceleration := 42000.0;
			axis.cmd := CONST.AXIS.STOP;
			StateCtrl := CTRL_SAFETYSTOP;
		END_IF

	CTRL_SAFETYSTOP:
		timer(PT := T#1600ms);
		IF BetrCtrl.value = CONST.MACHINEMODES.EMERGENCYSTOP THEN
			StateCtrl := CTRL_EMERGENCYSTOP_BEFORE;
		ELSE
			timer(IN := TRUE);
//			CASE state OF
//			ST_IDLE:
//				state := ST_QUIT;
//
//			ST_QUIT:
//				state := ST_QUIT;
//				axis.cmd := CONST.AXIS.RESET;
//				StateCtrl := CTRL_SAFETYSTOP_AFTER;
			IF  timer.Q THEN
				axis.cmd := CONST.AXIS.POWER_OFF;
				timer(IN := FALSE);
				StateCtrl := CTRL_SAFETYSTOP_AFTER;
			END_IF
	(*		END_CASE*)
		END_IF

	CTRL_SAFETYSTOP_AFTER:
		busy := FALSE;
		manualFirst := TRUE;
		status.ready := FALSE;
		IF BetrCtrl.value = CONST.MACHINEMODES.EMERGENCYSTOP THEN
			busy := TRUE;
			StateCtrl := CTRL_EMERGENCYSTOP_BEFORE;
		ELSIF BetrCtrl.value = CONST.MACHINEMODES.MANUAL THEN
				IF axis.MC_ReadStatus_0.Errorstop THEN
					axis.cmd := CONST.AXIS.RESET;
				END_IF
				supplydelay(IN:= TRUE, PT := T#8s);
				IF supplydelay.Q THEN
					axis.cmd := CONST.AXIS.POWER_ON;
					busy := TRUE;
					supplydelay(IN:= FALSE);
					StateCtrl := CTRL_MANUAL_BEFORE;
				END_IF
		ELSIF BetrCtrl.value = CONST.MACHINEMODES.AUTOMATIC  THEN
				IF axis.MC_ReadStatus_0.Errorstop THEN
					axis.cmd := CONST.AXIS.RESET;
				END_IF
				supplydelay(IN:= TRUE, PT := T#8s);
				IF supplydelay.Q THEN
					axis.cmd := CONST.AXIS.POWER_ON;
					busy := TRUE;
					supplydelay(IN:= FALSE);
					StateCtrl := CTRL_AUTO_BEFORE;
				END_IF

		END_IF

	CTRL_EMERGENCYSTOP_BEFORE:
		status.ready := FALSE;
		axis.cmd := CONST.AXIS.POWER_OFF;
		BetrStatus(set := TRUE, value := CONST.MACHINEMODES.EMERGENCYSTOP);
		busy := FALSE;
		StateCtrl := CTRL_EMERGENCYSTOP;

	CTRL_EMERGENCYSTOP:
		IF BetrCtrl.value = CONST.MACHINEMODES.EMERGENCYSTOP THEN
			;
		ELSE
			busy := TRUE;
			timer(IN := TRUE, PT := T#2s);
			StateCtrl := CTRL_EMERGENCYSTOP_AFTER;
		END_IF

	CTRL_EMERGENCYSTOP_AFTER:
		timer();
		IF BetrCtrl.value = CONST.MACHINEMODES.EMERGENCYSTOP THEN
			timer(IN := FALSE);
			BetrStatus(set := TRUE , value := CONST.MACHINEMODES.EMERGENCYSTOP);
			busy := FALSE;
			StateCtrl := CTRL_EMERGENCYSTOP;
		ELSIF timer.Q THEN
			timer(IN := FALSE);
			StateCtrl := CTRL_RESET_START;
		END_IF

	ELSE
		;
	END_CASE

	axis.BasicControl.Parameter.Deceleration	:= 20000.0; //only for initialization
	axis.BasicControl.Parameter.Acceleration	:= 20000.0;
//	gridwinderright.axis.BasicControl.Parameter.Deceleration:= 20000.0; //only for initialization
//	gridwinderright.axis.BasicControl.Parameter.Acceleration:= 20000.0;
//	feeder.BasicControl.Parameter.Acceleration := 20000;
//	feeder.BasicControl.Parameter.Deceleration := 20000;
END_FUNCTION_BLOCK
```

#### ac_manualGridWin.st
```iecst
(********************************************************************
 * COPYRIGHT -- Microsoft
 ********************************************************************
 * Programm: MAIN
 * Datei: ac_manualGridWin.st
 * Autor: awalz
 * Erstellt: 25. Juni 2014
 ********************************************************************
 * Implementierung des Programms MAIN
 ********************************************************************)

(* Fügt eine neue Aktion zum IEC Programm oder Bibliothek *)
ACTION ac_manualGridWin:
			CASE state OF

	ST_IDLE:
//		IF BetrCtrl.value <> CONST.MACHINEMODES.MANUAL THEN
//			state := ST_IDLE;
//			err(reset := TRUE);
//			busy := TRUE;
//			status.ready := FALSE;
//			StateCtrl := CTRL_MANUAL_AFTER;
//		ELSE
			IF axis.MC_ReadStatus_0.Error OR axis.MC_ReadStatus_0.Errorstop  THEN
				axis.cmd := CONST.AXIS.RESET;
				state := ST_AXIS_STOP;
			ELSE
				IF data.recipeData.mode = CONST.UNITMODEs.ENABLE THEN
					IF axis.MC_ReadStatus_0.Disabled THEN
						axis(cmd := CONST.AXIS.POWER_ON, machineaxis := machineaxis, data := data);
						state := ST_AXIS_ON;
					ELSIF axis.MC_ReadStatus_0.StandStill THEN
				(*		axis(cmd := CONST.AXIS.START, machineaxis := machineaxis, data := data);*)
						axis.cmd := CONST.AXIS.START;
						state := ST_AXIS_RUN;
					END_IF
				ELSIF data.recipeData.mode =  CONST.UNITMODEs.DISABLE THEN
					IF axis.MC_ReadStatus_0.Disabled THEN
						axis(cmd := CONST.AXIS.POWER_ON, machineaxis := machineaxis, data := data);
						state := ST_AXIS_ON_DIS;
					ELSE
						axis(cmd := CONST.AXIS.STOP, machineaxis := machineaxis, data := data);
						state := ST_AXIS_STOP;
					END_IF
				ELSIF data.recipeData.mode = CONST.UNITMODEs.AXIS_OFF THEN
					axis(cmd := CONST.AXIS.POWER_OFF, machineaxis := machineaxis, data := data);
					state := ST_AXIS_OFF;
				END_IF
			END_IF
//		END_IF

	ST_AXIS_STOP:
			IF data.recipeData.mode <> CONST.UNITMODEs.DISABLE THEN
				state := ST_IDLE;
/////////// wenn die Achse disable ist und die Maschine los läuft die Ache automatisch starten
			ELSIF machineaxis.MC_ReadStatus_0.ContinuousMotion THEN
				data.recipeData.mode :=  CONST.UNITMODEs.ENABLE;
				axis.cmd := CONST.AXIS.START;
				state := ST_IDLE;
			END_IF

	ST_AXIS_ON_DIS:
			IF data.recipeData.mode = CONST.UNITMODEs.DISABLE THEN
				state := ST_IDLE;
			END_IF

	ST_AXIS_RUN:
//			IF data.recipeData.mode <> CONST.UNITMODEs.ENABLE OR axis.MC_ReadStatus_0.Disabled OR axis.MC_ReadStatus_0.StandStill THEN
//				state := ST_IDLE;
//			END_IF
			IF data.recipeData.mode <> CONST.UNITMODEs.ENABLE (*OR NOT axis.MC_ReadStatus_0.ContinuousMotion*) THEN
				state := ST_IDLE;
			END_IF

	ST_AXIS_ON:

			IF data.recipeData.mode = CONST.UNITMODEs.ENABLE THEN
				state := ST_IDLE;
			ELSIF data.recipeData.mode	<> CONST.UNITMODEs.ENABLE AND axis.MC_ReadStatus_0.ContinuousMotion THEN
				state := ST_IDLE;
			END_IF

//			IF data.recipeData.mode <> CONST.UNITMODEs.ENABLE THEN
//				state := ST_IDLE;
//			END_IF

	ST_AXIS_OFF:
			IF data.recipeData.mode <> CONST.UNITMODEs.AXIS_OFF THEN
				state := ST_IDLE;
			END_IF

	END_CASE
END_ACTION
```

#### ac_TurnGridwinSetAfter.st
```iecst
(********************************************************************
 * COPYRIGHT -- Microsoft
 ********************************************************************
 * Programm: MAIN
 * Datei: ac_TurnGridwinSetafter.st
 * Autor: awalz
 * Erstellt: 25. Juni 2014
 ********************************************************************
 * Implementierung des Programms MAIN
 ********************************************************************)

(* Fügt eine neue Aktion zum IEC Programm oder Bibliothek *)
ACTION ac_TurnGridwinSetAfter:
	IF BetrCtrl.value = CONST.MACHINEMODES.EMERGENCYSTOP THEN
		StateCtrl := CTRL_EMERGENCYSTOP_BEFORE;
	ELSIF BetrCtrl.value = CONST.MACHINEMODES.SAFETYSTOP THEN
		StateCtrl := CTRL_SAFETYSTOP_BEFORE;
	ELSIF BetrCtrl.value = CONST.MACHINEMODES.MANUAL THEN
		StateCtrl := CTRL_STOP_BEFORE;
	ELSIF BetrCtrl.value = CONST.MACHINEMODES.AUTOMATIC THEN
		StateCtrl := CTRL_STOP_BEFORE;
	END_IF
END_ACTION
```

#### FB_GRIDWINDER.st
```iecst
(********************************************************************
 * COPYRIGHT -- Microsoft
 ********************************************************************
 * Programm: MAIN
 * Datei: FB_GRIDWINDER.st
 * Autor: awalz
 * Erstellt: 25. Juni 2014
 ********************************************************************
 * Implementierung des Programms MAIN
 ********************************************************************)

(* TODO: Bitte Kommentar hier einfügen *)
FUNCTION_BLOCK FB_GRIDWINDER
END_FUNCTION_BLOCK
```

#### Package Logical/MainMachineCtrl/MAIN/CuttingUnit - Neues leeres Paket
